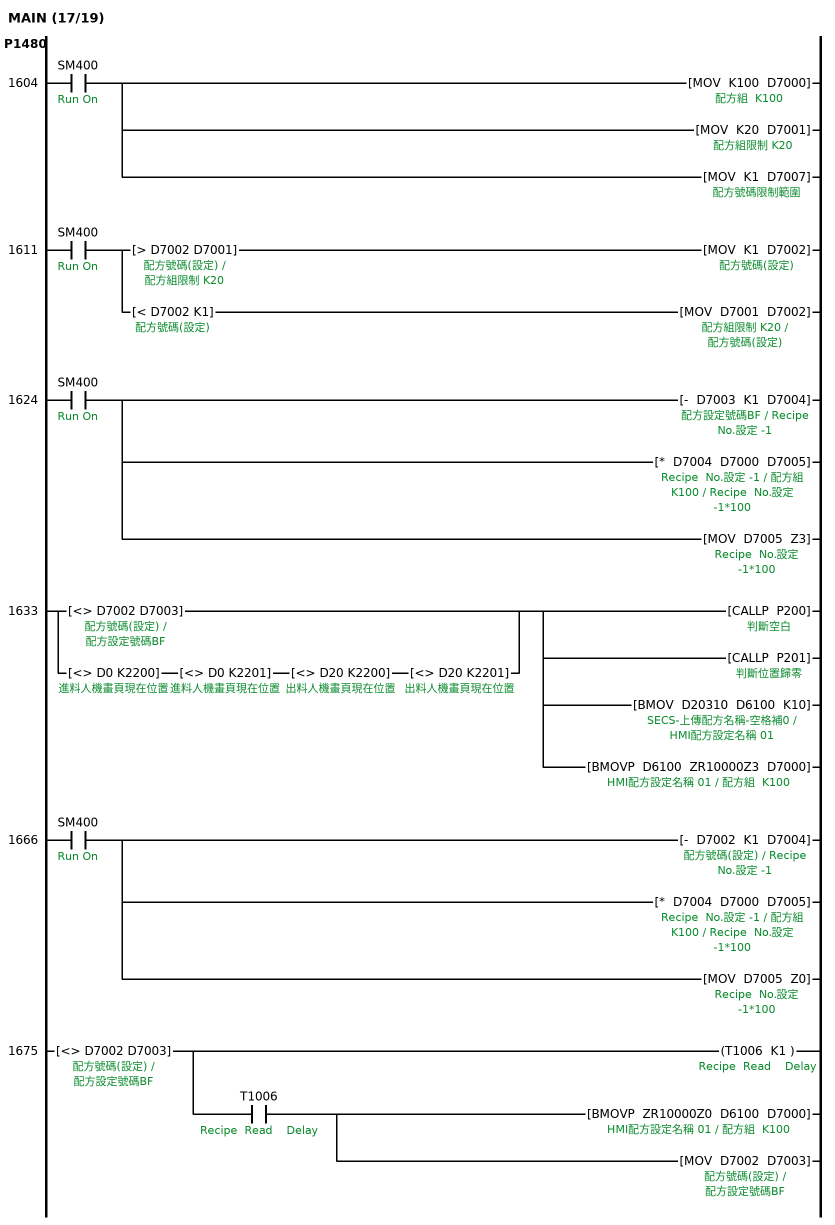
[picture p144: ladder of MAIN, rungs at steps 1604 to 1675]
1604  LD      SM400  ; Run On
      MOV     K100 D7000  ; 配方組  K100
      MOV     K20 D7001  ; 配方組限制 K20
      MOV     K1 D7007  ; 配方號碼限制範圍
1611  LD      SM400  ; Run On
      MPS
      AND>    D7002 D7001  ; 配方號碼(設定) / 配方組限制 K20
      MOV     K1 D7002
      MPP
      AND<    D7002 K1  ; 配方號碼(設定)
      MOV     D7001 D7002
1624  LD      SM400  ; Run On
      -       D7003 K1 D7004  ; 配方設定號碼BF / Recipe  No.設定 -1
      *       D7004 D7000 D7005  ; Recipe  No.設定 -1*100
      MOV     D7005 Z3
1633  LD<>    D7002 D7003  ; 配方號碼(設定) / 配方設定號碼BF
      LD<>    D0 K2200  ; 進料人機畫頁現在位置
      AND<>   D0 K2201  ; 進料人機畫頁現在位置
      AND<>   D20 K2200  ; 出料人機畫頁現在位置
      AND<>   D20 K2201  ; 出料人機畫頁現在位置
      ORB
      CALLP   P200  ; 判斷空白
      CALLP   P201  ; 判斷位置歸零
      BMOV    D20310 D6100 K10  ; SECS-上傳配方名稱-空格補0 / HMI配方設定名稱 01
      BMOVP   D6100 ZR10000Z3 D7000
1666  LD      SM400  ; Run On
      -       D7002 K1 D7004
      *       D7004 D7000 D7005
      MOV     D7005 Z0
1675  LD<>    D7002 D7003  ; 配方號碼(設定) / 配方設定號碼BF
      OUT     T1006 K1  ; Recipe  Read    Delay
      AND     T1006  ; Recipe  Read    Delay
      BMOVP   ZR10000Z0 D6100 D7000
      MOV     D7002 D7003
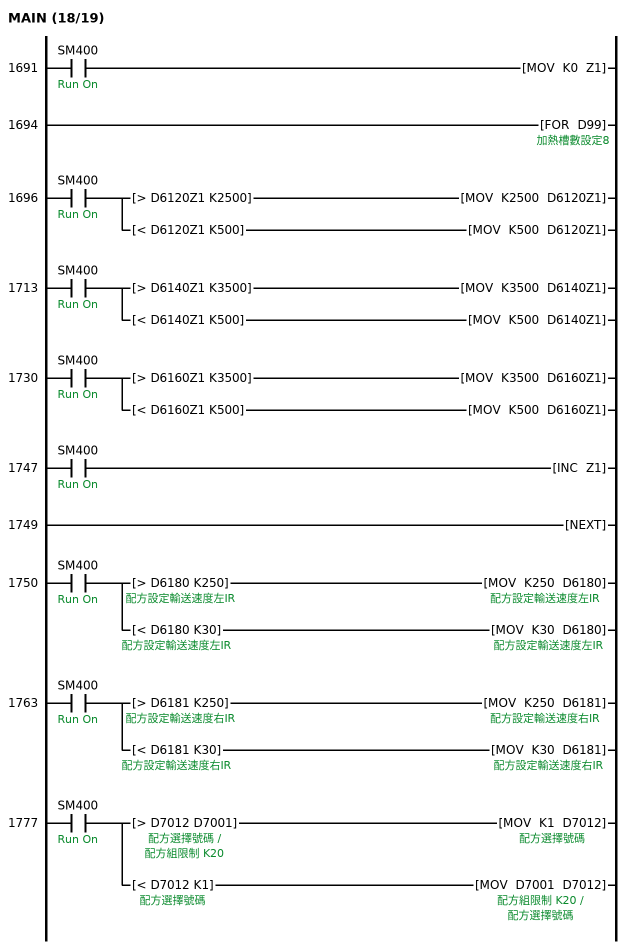
1691  LD      SM400  ; Run On
      MOV     K0 Z1
1694  FOR     D99
1696  LD      SM400  ; Run On
      MPS
      AND>    D6120Z1 K2500
      MOV     K2500 D6120Z1
      MPP
      AND<    D6120Z1 K500
      MOV     K500 D6120Z1
1713  LD      SM400  ; Run On
      MPS
      AND>    D6140Z1 K3500
      MOV     K3500 D6140Z1
      MPP
      AND<    D6140Z1 K500
      MOV     K500 D6140Z1
1730  LD      SM400  ; Run On
      MPS
      AND>    D6160Z1 K3500
      MOV     K3500 D6160Z1
      MPP
      AND<    D6160Z1 K500
      MOV     K500 D6160Z1
1747  LD      SM400  ; Run On
      INC     Z1
1749  NEXT
1750  LD      SM400  ; Run On
      MPS
      AND>    D6180 K250  ; 配方設定輸送速度左IR
      MOV     K250 D6180
      MPP
      AND<    D6180 K30  ; 配方設定輸送速度左IR
      MOV     K30 D6180
1763  LD      SM400  ; Run On
      MPS
      AND>    D6181 K250  ; 配方設定輸送速度右IR
      MOV     K250 D6181
      MPP
      AND<    D6181 K30  ; 配方設定輸送速度右IR
      MOV     K30 D6181
1777  LD      SM400  ; Run On
      MPS
      AND>    D7012 D7001  ; 配方選擇號碼 / 配方組限制 K20
      MOV     K1 D7012
      MPP
      AND<    D7012 K1  ; 配方選擇號碼
      MOV     D7001 D7012
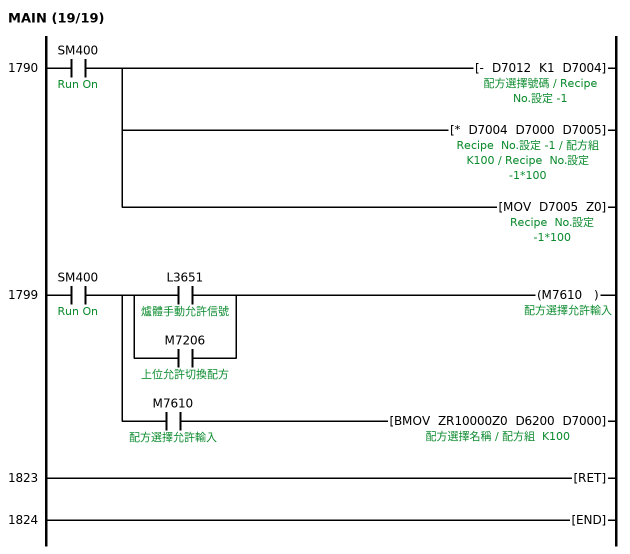
1790  LD      SM400  ; Run On
      -       D7012 K1 D7004
      *       D7004 D7000 D7005
      MOV     D7005 Z0
1799  LD      SM400  ; Run On
      MPS
      LD      L3651  ; 爐體手動允許信號
      OR      M7206  ; 上位允許切換配方
      ANB
      OUT     M7610  ; 配方選擇允許輸入
      MPP
      AND     M7610  ; 配方選擇允許輸入
      BMOV    ZR10000Z0 D6200 D7000  ; 配方選擇名稱
        [note] /* 配方選擇切換 */
1823  RET
1824  END
END_PROGRAM

PROGRAM HEAT
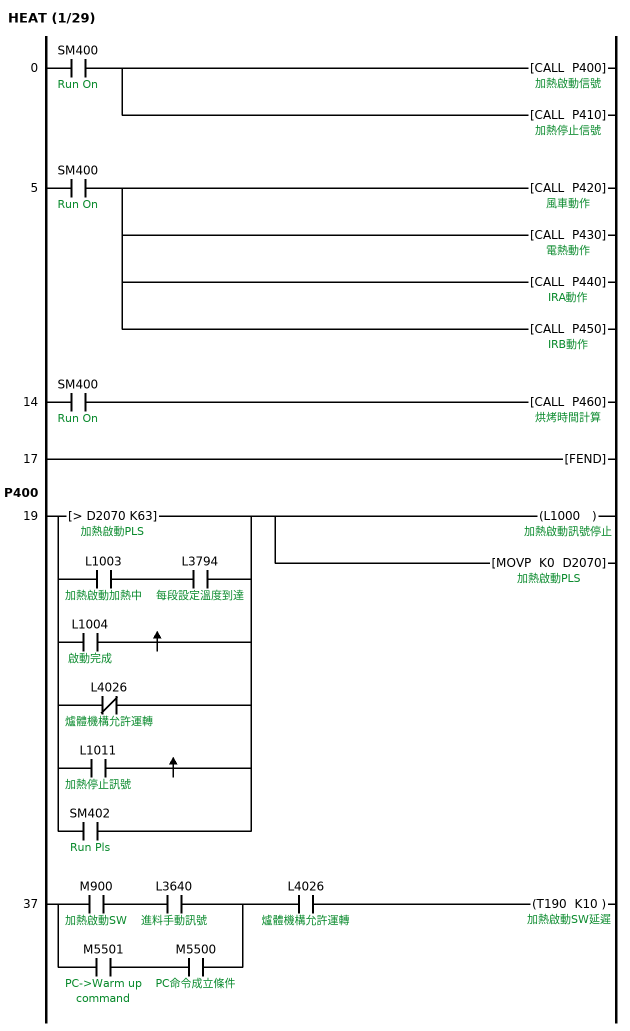
0     LD      SM400  ; Run On
      CALL    P400  ; 加熱啟動信號
      CALL    P410  ; 加熱停止信號
5     LD      SM400  ; Run On
      CALL    P420  ; 風車動作
      CALL    P430  ; 電熱動作
      CALL    P440  ; IRA動作
      CALL    P450  ; IRB動作
14    LD      SM400  ; Run On
      CALL    P460  ; 烘烤時間計算
17    FEND
      P400
19    LD>     D2070 K63  ; 加熱啟動PLS
      LD      L1003  ; 加熱啟動加熱中
      AND     L3794  ; 每段設定溫度到達
      ORB
      LD      L1004  ; 啟動完成
      MEP
      ORB
      ORI     L4026  ; 爐體機構允許運轉
      LD      L1011  ; 加熱停止訊號
      MEP
      ORB
      OR      SM402  ; Run Pls
      OUT     L1000  ; 加熱啟動訊號停止
      MOVP    K0 D2070
37    LD      M900  ; 加熱啟動SW
      AND     L3640  ; 進料手動訊號
      LD      M5501  ; PC->Warm up command
      AND     M5500  ; PC命令成立條件
      ORB
      AND     L4026  ; 爐體機構允許運轉
      OUT     T190 K10  ; 加熱啟動SW延遲
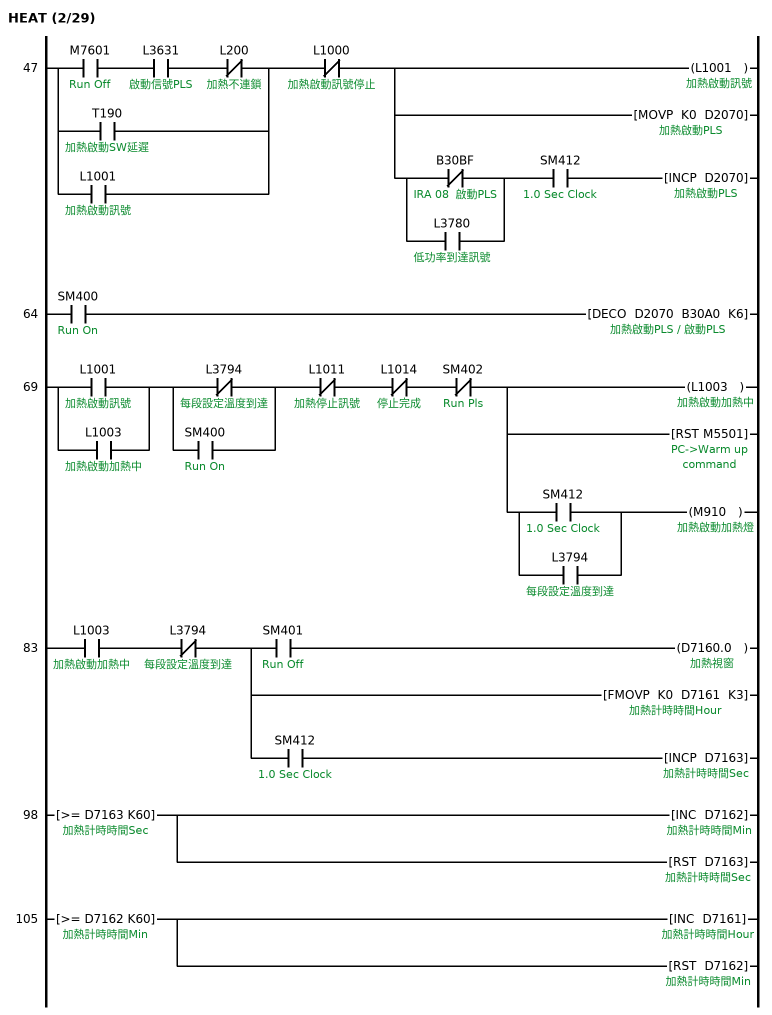
47    LD      M7601  ; Run Off
      AND     L3631  ; 啟動信號PLS
      ANI     L200  ; 加熱不連鎖
      OR      T190  ; 加熱啟動SW延遲
      OR      L1001  ; 加熱啟動訊號
      ANI     L1000  ; 加熱啟動訊號停止
      OUT     L1001  ; 加熱啟動訊號
      MOVP    K0 D2070
      LDI     B30BF  ; IRA 08  啟動PLS
      OR      L3780  ; 低功率到達訊號
      ANB
      AND     SM412  ; 1.0 Sec Clock
      INCP    D2070
64    LD      SM400  ; Run On
      DECO    D2070 B30A0 K6  ; 啟動PLS
69    LD      L1001  ; 加熱啟動訊號
      OR      L1003  ; 加熱啟動加熱中
      LDI     L3794  ; 每段設定溫度到達
      OR      SM400  ; Run On
      ANB
      ANI     L1011  ; 加熱停止訊號
      ANI     L1014  ; 停止完成
      ANI     SM402  ; Run Pls
      OUT     L1003  ; 加熱啟動加熱中
      RST     M5501  ; PC->Warm up command
      LD      SM412  ; 1.0 Sec Clock
      OR      L3794  ; 每段設定溫度到達
      ANB
      OUT     M910  ; 加熱啟動加熱燈
83    LD      L1003  ; 加熱啟動加熱中
      ANI     L3794  ; 每段設定溫度到達
      MPS
      AND     SM401  ; Run Off
      OUT     D7160.0  ; 加熱視窗
      MPP
      FMOVP   K0 D7161 K3  ; 加熱計時時間Hour
      AND     SM412  ; 1.0 Sec Clock
      INCP    D7163  ; 加熱計時時間Sec
98    LD>=    D7163 K60  ; 加熱計時時間Sec
      INC     D7162  ; 加熱計時時間Min
      RST     D7163  ; 加熱計時時間Sec
105   LD>=    D7162 K60  ; 加熱計時時間Min
      INC     D7161
      RST     D7162  ; 加熱計時時間Min
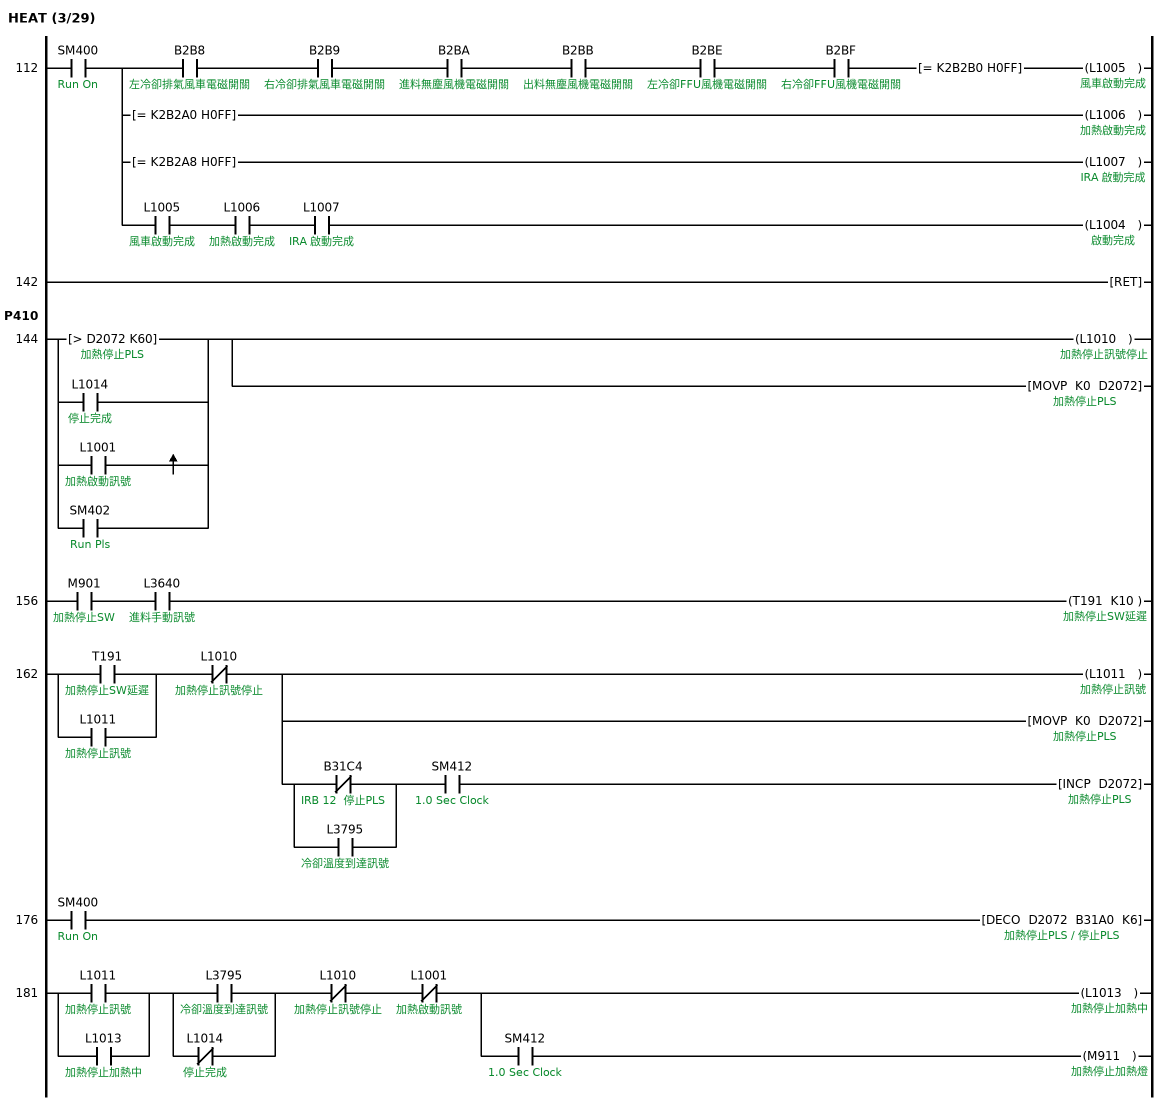
112   LD      SM400  ; Run On
      MPS
      AND     B2B8  ; 左冷卻排氣風車電磁開關
      AND     B2B9  ; 右冷卻排氣風車電磁開關
      AND     B2BA  ; 進料無塵風機電磁開關
      AND     B2BB  ; 出料無塵風機電磁開關
      AND     B2BE  ; 左冷卻FFU風機電磁開關
      AND     B2BF  ; 右冷卻FFU風機電磁開關
      AND=    K2B2B0 H0FF  ; 第01槽風車電磁開關
      OUT     L1005  ; 風車啟動完成
      MRD
      AND=    K2B2A0 H0FF  ; 第01槽熱風H01電磁開關
      OUT     L1006  ; 加熱啟動完成
      MRD
      AND=    K2B2A8 H0FF  ; 第01槽IR01A電磁開關
      OUT     L1007  ; IRA 啟動完成
      MPP
      AND     L1005  ; 風車啟動完成
      AND     L1006  ; 加熱啟動完成
      AND     L1007  ; IRA 啟動完成
      OUT     L1004  ; 啟動完成
142   RET
      P410
144   LD>     D2072 K60  ; 加熱停止PLS
      OR      L1014  ; 停止完成
      LD      L1001  ; 加熱啟動訊號
      MEP
      ORB
      OR      SM402  ; Run Pls
      OUT     L1010  ; 加熱停止訊號停止
      MOVP    K0 D2072
156   LD      M901  ; 加熱停止SW
      AND     L3640  ; 進料手動訊號
      OUT     T191 K10  ; 加熱停止SW延遲
162   LD      T191  ; 加熱停止SW延遲
      OR      L1011  ; 加熱停止訊號
      ANI     L1010  ; 加熱停止訊號停止
      OUT     L1011  ; 加熱停止訊號
      MOVP    K0 D2072
      LDI     B31C4  ; IRB 12  停止PLS
      OR      L3795  ; 冷卻溫度到達訊號
      ANB
      AND     SM412  ; 1.0 Sec Clock
      INCP    D2072
176   LD      SM400  ; Run On
      DECO    D2072 B31A0 K6  ; 停止PLS
181   LD      L1011  ; 加熱停止訊號
      OR      L1013  ; 加熱停止加熱中
      LD      L3795  ; 冷卻溫度到達訊號
      ORI     L1014  ; 停止完成
      ANB
      ANI     L1010  ; 加熱停止訊號停止
      ANI     L1001  ; 加熱啟動訊號
      OUT     L1013  ; 加熱停止加熱中
      AND     SM412  ; 1.0 Sec Clock
      OUT     M911  ; 加熱停止加熱燈
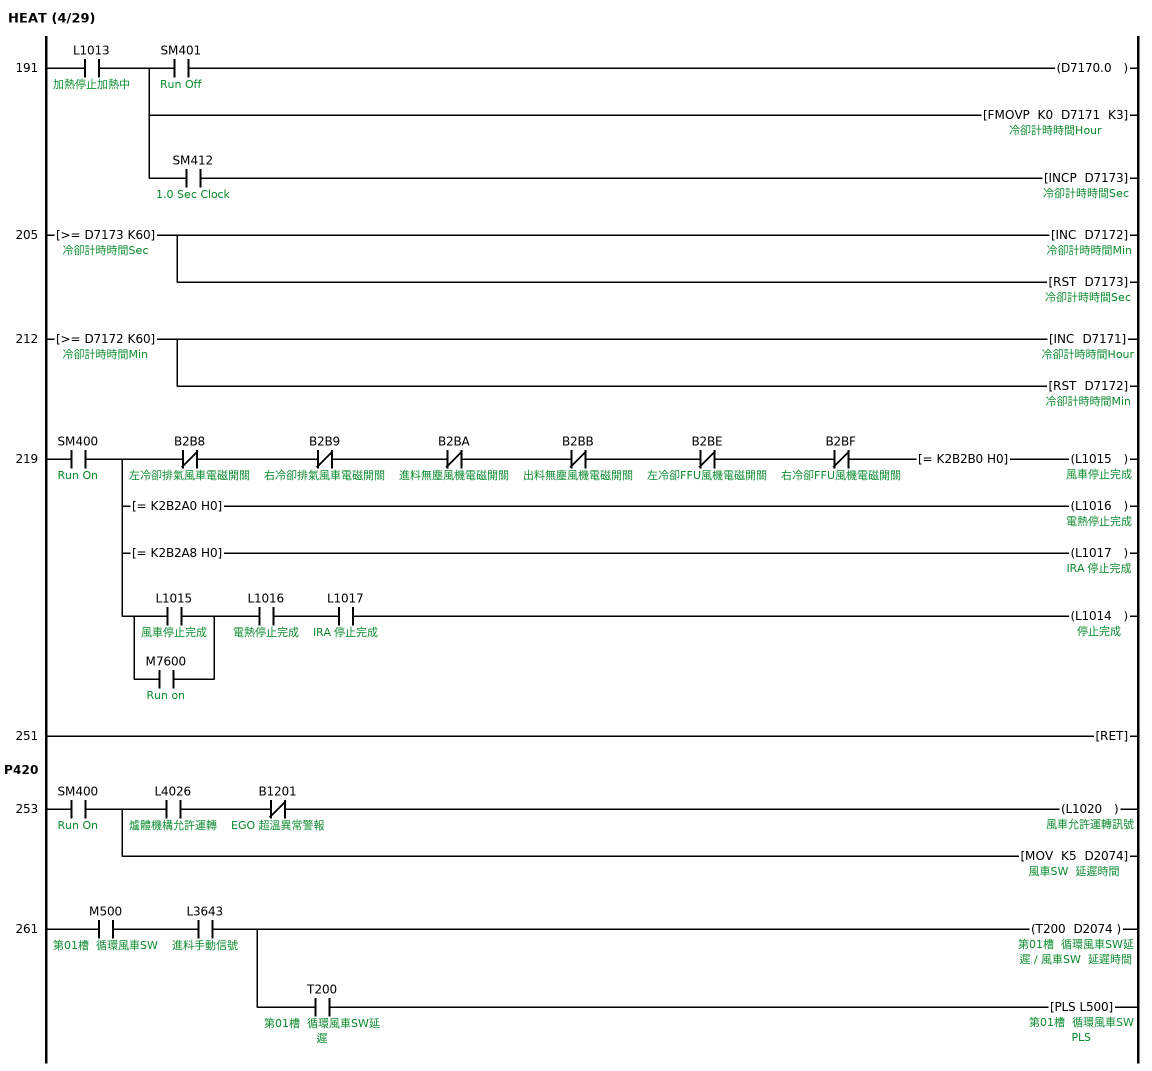
191   LD      L1013  ; 加熱停止加熱中
      MPS
      AND     SM401  ; Run Off
      OUT     D7170.0
      MPP
      FMOVP   K0 D7171 K3  ; 冷卻計時時間Hour
      AND     SM412  ; 1.0 Sec Clock
      INCP    D7173  ; 冷卻計時時間Sec
205   LD>=    D7173 K60  ; 冷卻計時時間Sec
      INC     D7172  ; 冷卻計時時間Min
      RST     D7173  ; 冷卻計時時間Sec
212   LD>=    D7172 K60  ; 冷卻計時時間Min
      INC     D7171
      RST     D7172  ; 冷卻計時時間Min
219   LD      SM400  ; Run On
      MPS
      ANI     B2B8  ; 左冷卻排氣風車電磁開關
      ANI     B2B9  ; 右冷卻排氣風車電磁開關
      ANI     B2BA  ; 進料無塵風機電磁開關
      ANI     B2BB  ; 出料無塵風機電磁開關
      ANI     B2BE  ; 左冷卻FFU風機電磁開關
      ANI     B2BF  ; 右冷卻FFU風機電磁開關
      AND=    K2B2B0 H0  ; 第01槽風車電磁開關
      OUT     L1015  ; 風車停止完成
      MRD
      AND=    K2B2A0 H0  ; 第01槽熱風H01電磁開關
      OUT     L1016  ; 電熱停止完成
      MRD
      AND=    K2B2A8 H0  ; 第01槽IR01A電磁開關
      OUT     L1017  ; IRA 停止完成
      MPP
      LD      L1015  ; 風車停止完成
      OR      M7600  ; Run on
      ANB
      AND     L1016  ; 電熱停止完成
      AND     L1017  ; IRA 停止完成
      OUT     L1014  ; 停止完成
251   RET
      P420
253   LD      SM400  ; Run On
      MPS
      AND     L4026  ; 爐體機構允許運轉
      ANI     B1201  ; EGO 超溫異常警報
      OUT     L1020  ; 風車允許運轉訊號
      MPP
      MOV     K5 D2074  ; 風車SW  延遲時間
261   LD      M500  ; 第01槽  循環風車SW
      AND     L3643  ; 進料手動信號
      OUT     T200 D2074  ; 第01槽  循環風車SW延遲 / 風車SW  延遲時間
      AND     T200  ; 第01槽  循環風車SW延遲
      PLS     L500  ; 第01槽  循環風車SW  PLS
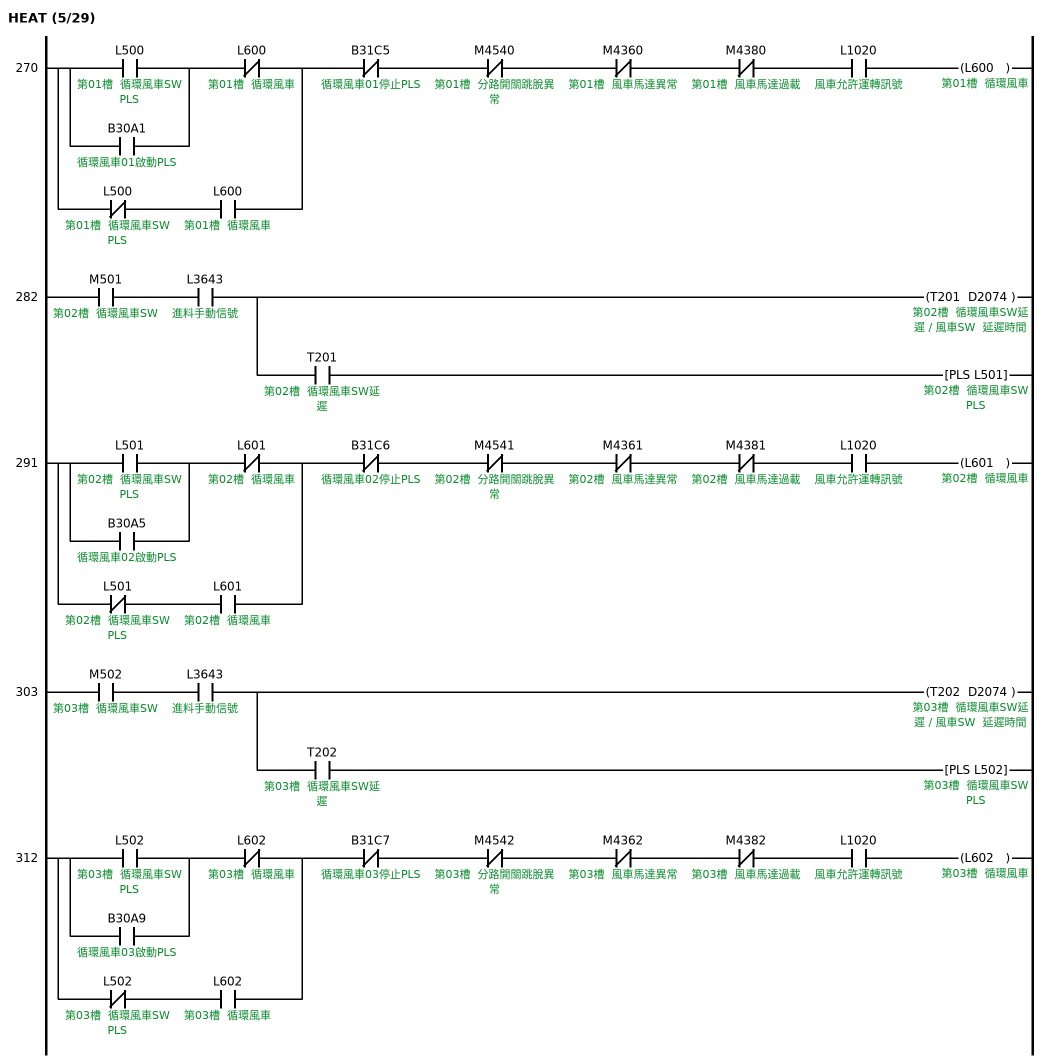
270   LD      L500  ; 第01槽  循環風車SW  PLS
      OR      B30A1  ; 循環風車01啟動PLS
      ANI     L600  ; 第01槽  循環風車
      LDI     L500  ; 第01槽  循環風車SW  PLS
      AND     L600  ; 第01槽  循環風車
      ORB
      ANI     B31C5  ; 循環風車01停止PLS
      ANI     M4540  ; 第01槽  分路開關跳脫異常
      ANI     M4360  ; 第01槽  風車馬達異常
      ANI     M4380  ; 第01槽  風車馬達過載
      AND     L1020  ; 風車允許運轉訊號
      OUT     L600  ; 第01槽  循環風車
282   LD      M501  ; 第02槽  循環風車SW
      AND     L3643  ; 進料手動信號
      OUT     T201 D2074  ; 第02槽  循環風車SW延遲 / 風車SW  延遲時間
      AND     T201  ; 第02槽  循環風車SW延遲
      PLS     L501  ; 第02槽  循環風車SW  PLS
291   LD      L501  ; 第02槽  循環風車SW  PLS
      OR      B30A5  ; 循環風車02啟動PLS
      ANI     L601  ; 第02槽  循環風車
      LDI     L501  ; 第02槽  循環風車SW  PLS
      AND     L601  ; 第02槽  循環風車
      ORB
      ANI     B31C6  ; 循環風車02停止PLS
      ANI     M4541  ; 第02槽  分路開關跳脫異常
      ANI     M4361  ; 第02槽  風車馬達異常
      ANI     M4381  ; 第02槽  風車馬達過載
      AND     L1020  ; 風車允許運轉訊號
      OUT     L601  ; 第02槽  循環風車
303   LD      M502  ; 第03槽  循環風車SW
      AND     L3643  ; 進料手動信號
      OUT     T202 D2074  ; 第03槽  循環風車SW延遲 / 風車SW  延遲時間
      AND     T202  ; 第03槽  循環風車SW延遲
      PLS     L502  ; 第03槽  循環風車SW  PLS
312   LD      L502  ; 第03槽  循環風車SW  PLS
      OR      B30A9  ; 循環風車03啟動PLS
      ANI     L602  ; 第03槽  循環風車
      LDI     L502  ; 第03槽  循環風車SW  PLS
      AND     L602  ; 第03槽  循環風車
      ORB
      ANI     B31C7  ; 循環風車03停止PLS
      ANI     M4542  ; 第03槽  分路開關跳脫異常
      ANI     M4362  ; 第03槽  風車馬達異常
      ANI     M4382  ; 第03槽  風車馬達過載
      AND     L1020  ; 風車允許運轉訊號
      OUT     L602  ; 第03槽  循環風車
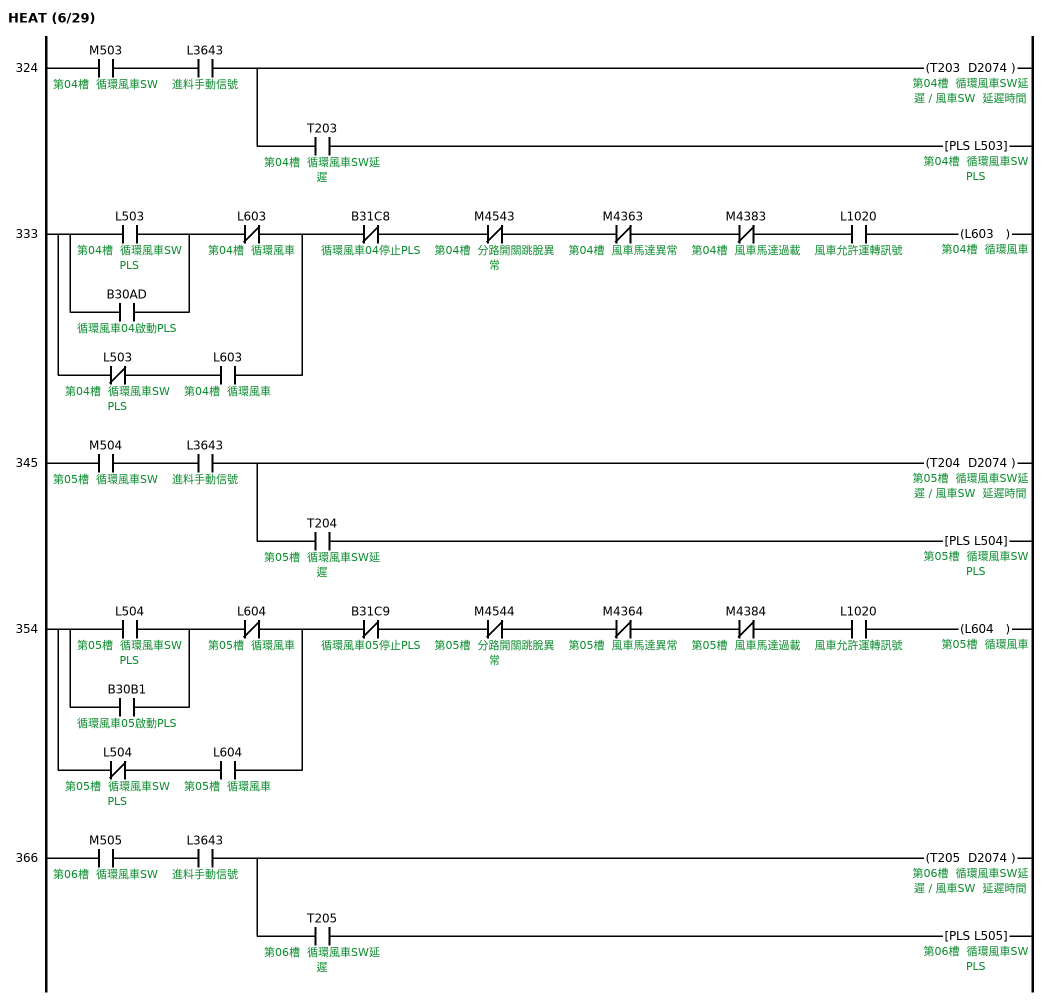
324   LD      M503  ; 第04槽  循環風車SW
      AND     L3643  ; 進料手動信號
      OUT     T203 D2074  ; 第04槽  循環風車SW延遲 / 風車SW  延遲時間
      AND     T203  ; 第04槽  循環風車SW延遲
      PLS     L503  ; 第04槽  循環風車SW  PLS
333   LD      L503  ; 第04槽  循環風車SW  PLS
      OR      B30AD  ; 循環風車04啟動PLS
      ANI     L603  ; 第04槽  循環風車
      LDI     L503  ; 第04槽  循環風車SW  PLS
      AND     L603  ; 第04槽  循環風車
      ORB
      ANI     B31C8  ; 循環風車04停止PLS
      ANI     M4543  ; 第04槽  分路開關跳脫異常
      ANI     M4363  ; 第04槽  風車馬達異常
      ANI     M4383  ; 第04槽  風車馬達過載
      AND     L1020  ; 風車允許運轉訊號
      OUT     L603  ; 第04槽  循環風車
345   LD      M504  ; 第05槽  循環風車SW
      AND     L3643  ; 進料手動信號
      OUT     T204 D2074  ; 第05槽  循環風車SW延遲 / 風車SW  延遲時間
      AND     T204  ; 第05槽  循環風車SW延遲
      PLS     L504  ; 第05槽  循環風車SW  PLS
354   LD      L504  ; 第05槽  循環風車SW  PLS
      OR      B30B1  ; 循環風車05啟動PLS
      ANI     L604  ; 第05槽  循環風車
      LDI     L504  ; 第05槽  循環風車SW  PLS
      AND     L604  ; 第05槽  循環風車
      ORB
      ANI     B31C9  ; 循環風車05停止PLS
      ANI     M4544  ; 第05槽  分路開關跳脫異常
      ANI     M4364  ; 第05槽  風車馬達異常
      ANI     M4384  ; 第05槽  風車馬達過載
      AND     L1020  ; 風車允許運轉訊號
      OUT     L604  ; 第05槽  循環風車
366   LD      M505  ; 第06槽  循環風車SW
      AND     L3643  ; 進料手動信號
      OUT     T205 D2074  ; 第06槽  循環風車SW延遲 / 風車SW  延遲時間
      AND     T205  ; 第06槽  循環風車SW延遲
      PLS     L505  ; 第06槽  循環風車SW  PLS
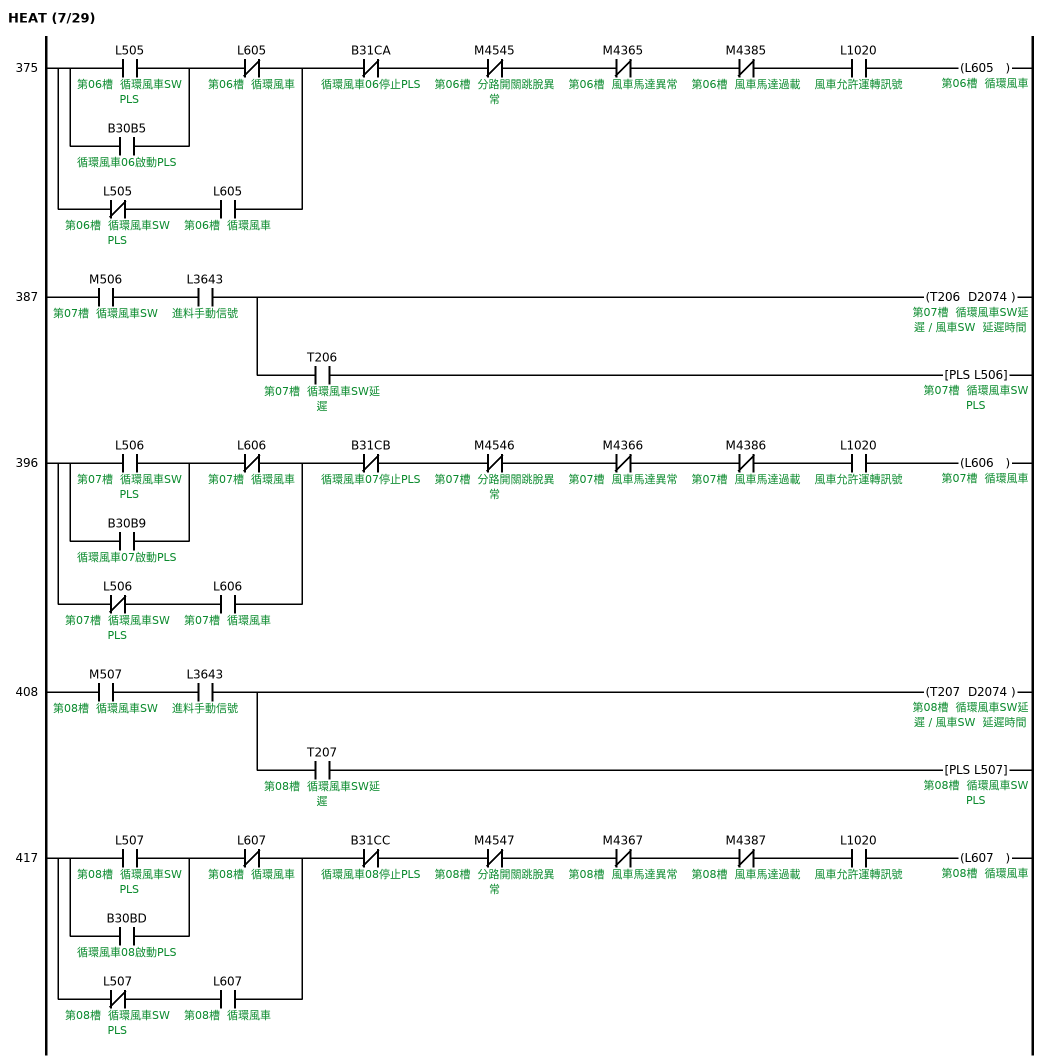
375   LD      L505  ; 第06槽  循環風車SW  PLS
      OR      B30B5  ; 循環風車06啟動PLS
      ANI     L605  ; 第06槽  循環風車
      LDI     L505  ; 第06槽  循環風車SW  PLS
      AND     L605  ; 第06槽  循環風車
      ORB
      ANI     B31CA  ; 循環風車06停止PLS
      ANI     M4545  ; 第06槽  分路開關跳脫異常
      ANI     M4365  ; 第06槽  風車馬達異常
      ANI     M4385  ; 第06槽  風車馬達過載
      AND     L1020  ; 風車允許運轉訊號
      OUT     L605  ; 第06槽  循環風車
387   LD      M506  ; 第07槽  循環風車SW
      AND     L3643  ; 進料手動信號
      OUT     T206 D2074  ; 第07槽  循環風車SW延遲 / 風車SW  延遲時間
      AND     T206  ; 第07槽  循環風車SW延遲
      PLS     L506  ; 第07槽  循環風車SW  PLS
396   LD      L506  ; 第07槽  循環風車SW  PLS
      OR      B30B9  ; 循環風車07啟動PLS
      ANI     L606  ; 第07槽  循環風車
      LDI     L506  ; 第07槽  循環風車SW  PLS
      AND     L606  ; 第07槽  循環風車
      ORB
      ANI     B31CB  ; 循環風車07停止PLS
      ANI     M4546  ; 第07槽  分路開關跳脫異常
      ANI     M4366  ; 第07槽  風車馬達異常
      ANI     M4386  ; 第07槽  風車馬達過載
      AND     L1020  ; 風車允許運轉訊號
      OUT     L606  ; 第07槽  循環風車
408   LD      M507  ; 第08槽  循環風車SW
      AND     L3643  ; 進料手動信號
      OUT     T207 D2074  ; 第08槽  循環風車SW延遲 / 風車SW  延遲時間
      AND     T207  ; 第08槽  循環風車SW延遲
      PLS     L507  ; 第08槽  循環風車SW  PLS
417   LD      L507  ; 第08槽  循環風車SW  PLS
      OR      B30BD  ; 循環風車08啟動PLS
      ANI     L607  ; 第08槽  循環風車
      LDI     L507  ; 第08槽  循環風車SW  PLS
      AND     L607  ; 第08槽  循環風車
      ORB
      ANI     B31CC  ; 循環風車08停止PLS
      ANI     M4547  ; 第08槽  分路開關跳脫異常
      ANI     M4367  ; 第08槽  風車馬達異常
      ANI     M4387  ; 第08槽  風車馬達過載
      AND     L1020  ; 風車允許運轉訊號
      OUT     L607  ; 第08槽  循環風車
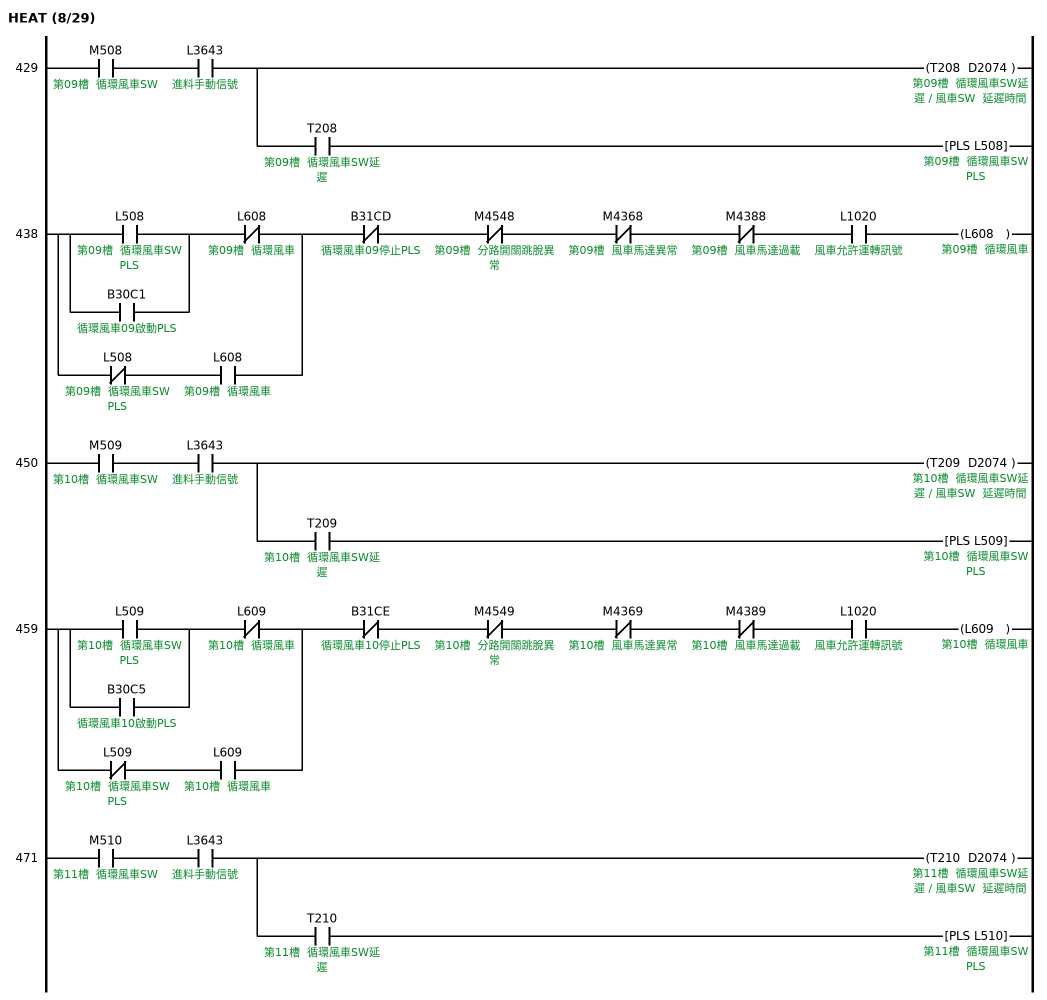
429   LD      M508  ; 第09槽  循環風車SW
      AND     L3643  ; 進料手動信號
      OUT     T208 D2074  ; 第09槽  循環風車SW延遲 / 風車SW  延遲時間
      AND     T208  ; 第09槽  循環風車SW延遲
      PLS     L508  ; 第09槽  循環風車SW  PLS
438   LD      L508  ; 第09槽  循環風車SW  PLS
      OR      B30C1  ; 循環風車09啟動PLS
      ANI     L608  ; 第09槽  循環風車
      LDI     L508  ; 第09槽  循環風車SW  PLS
      AND     L608  ; 第09槽  循環風車
      ORB
      ANI     B31CD  ; 循環風車09停止PLS
      ANI     M4548  ; 第09槽  分路開關跳脫異常
      ANI     M4368  ; 第09槽  風車馬達異常
      ANI     M4388  ; 第09槽  風車馬達過載
      AND     L1020  ; 風車允許運轉訊號
      OUT     L608  ; 第09槽  循環風車
450   LD      M509  ; 第10槽  循環風車SW
      AND     L3643  ; 進料手動信號
      OUT     T209 D2074  ; 第10槽  循環風車SW延遲 / 風車SW  延遲時間
      AND     T209  ; 第10槽  循環風車SW延遲
      PLS     L509  ; 第10槽  循環風車SW  PLS
459   LD      L509  ; 第10槽  循環風車SW  PLS
      OR      B30C5  ; 循環風車10啟動PLS
      ANI     L609  ; 第10槽  循環風車
      LDI     L509  ; 第10槽  循環風車SW  PLS
      AND     L609  ; 第10槽  循環風車
      ORB
      ANI     B31CE  ; 循環風車10停止PLS
      ANI     M4549  ; 第10槽  分路開關跳脫異常
      ANI     M4369  ; 第10槽  風車馬達異常
      ANI     M4389  ; 第10槽  風車馬達過載
      AND     L1020  ; 風車允許運轉訊號
      OUT     L609  ; 第10槽  循環風車
471   LD      M510  ; 第11槽  循環風車SW
      AND     L3643  ; 進料手動信號
      OUT     T210 D2074  ; 第11槽  循環風車SW延遲 / 風車SW  延遲時間
      AND     T210  ; 第11槽  循環風車SW延遲
      PLS     L510  ; 第11槽  循環風車SW  PLS
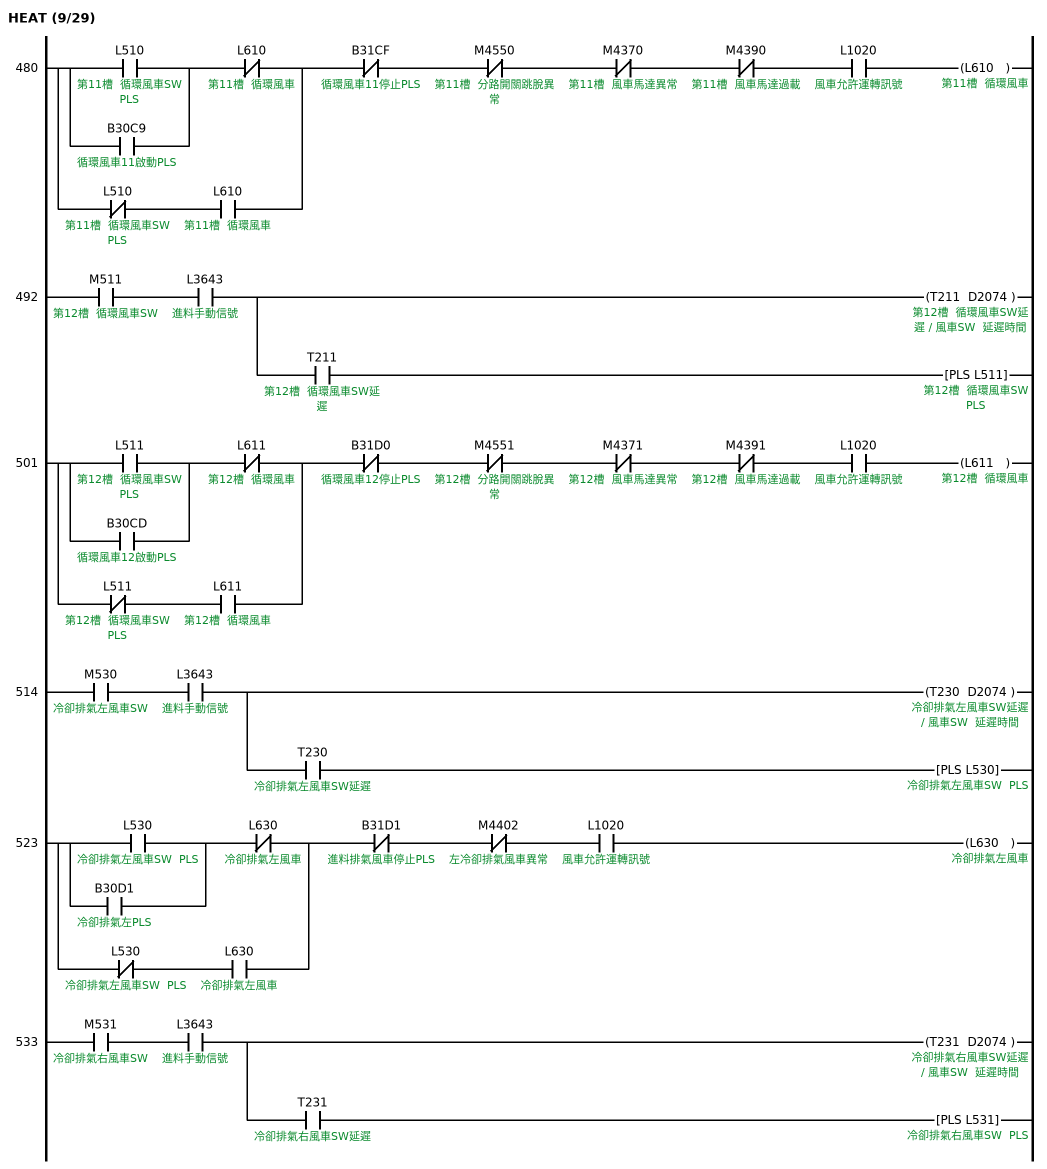
480   LD      L510  ; 第11槽  循環風車SW  PLS
      OR      B30C9  ; 循環風車11啟動PLS
      ANI     L610  ; 第11槽  循環風車
      LDI     L510  ; 第11槽  循環風車SW  PLS
      AND     L610  ; 第11槽  循環風車
      ORB
      ANI     B31CF  ; 循環風車11停止PLS
      ANI     M4550  ; 第11槽  分路開關跳脫異常
      ANI     M4370  ; 第11槽  風車馬達異常
      ANI     M4390  ; 第11槽  風車馬達過載
      AND     L1020  ; 風車允許運轉訊號
      OUT     L610  ; 第11槽  循環風車
492   LD      M511  ; 第12槽  循環風車SW
      AND     L3643  ; 進料手動信號
      OUT     T211 D2074  ; 第12槽  循環風車SW延遲 / 風車SW  延遲時間
      AND     T211  ; 第12槽  循環風車SW延遲
      PLS     L511  ; 第12槽  循環風車SW  PLS
501   LD      L511  ; 第12槽  循環風車SW  PLS
      OR      B30CD  ; 循環風車12啟動PLS
      ANI     L611  ; 第12槽  循環風車
      LDI     L511  ; 第12槽  循環風車SW  PLS
      AND     L611  ; 第12槽  循環風車
      ORB
      ANI     B31D0  ; 循環風車12停止PLS
      ANI     M4551  ; 第12槽  分路開關跳脫異常
      ANI     M4371  ; 第12槽  風車馬達異常
      ANI     M4391  ; 第12槽  風車馬達過載
      AND     L1020  ; 風車允許運轉訊號
      OUT     L611  ; 第12槽  循環風車
514   LD      M530  ; 冷卻排氣左風車SW
      AND     L3643  ; 進料手動信號
      OUT     T230 D2074  ; 冷卻排氣左風車SW延遲 / 風車SW  延遲時間
      AND     T230  ; 冷卻排氣左風車SW延遲
      PLS     L530  ; 冷卻排氣左風車SW  PLS
523   LD      L530  ; 冷卻排氣左風車SW  PLS
      OR      B30D1  ; 冷卻排氣左PLS
      ANI     L630  ; 冷卻排氣左風車
      LDI     L530  ; 冷卻排氣左風車SW  PLS
      AND     L630  ; 冷卻排氣左風車
      ORB
      ANI     B31D1  ; 進料排氣風車停止PLS
      ANI     M4402  ; 左冷卻排氣風車異常
      AND     L1020  ; 風車允許運轉訊號
      OUT     L630  ; 冷卻排氣左風車
533   LD      M531  ; 冷卻排氣右風車SW
      AND     L3643  ; 進料手動信號
      OUT     T231 D2074  ; 冷卻排氣右風車SW延遲 / 風車SW  延遲時間
      AND     T231  ; 冷卻排氣右風車SW延遲
      PLS     L531  ; 冷卻排氣右風車SW  PLS
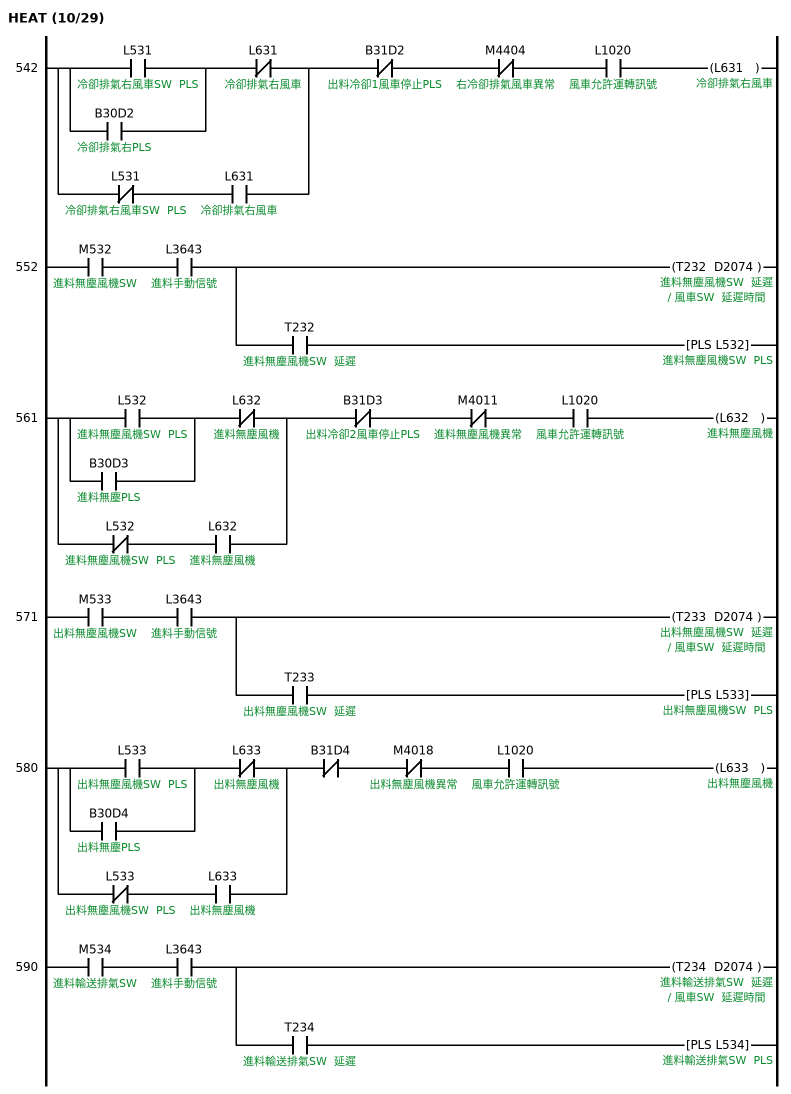
542   LD      L531  ; 冷卻排氣右風車SW  PLS
      OR      B30D2  ; 冷卻排氣右PLS
      ANI     L631  ; 冷卻排氣右風車
      LDI     L531  ; 冷卻排氣右風車SW  PLS
      AND     L631  ; 冷卻排氣右風車
      ORB
      ANI     B31D2  ; 出料冷卻1風車停止PLS
      ANI     M4404  ; 右冷卻排氣風車異常
      AND     L1020  ; 風車允許運轉訊號
      OUT     L631  ; 冷卻排氣右風車
552   LD      M532  ; 進料無塵風機SW
      AND     L3643  ; 進料手動信號
      OUT     T232 D2074  ; 進料無塵風機SW  延遲 / 風車SW  延遲時間
      AND     T232  ; 進料無塵風機SW  延遲
      PLS     L532  ; 進料無塵風機SW  PLS
561   LD      L532  ; 進料無塵風機SW  PLS
      OR      B30D3  ; 進料無塵PLS
      ANI     L632  ; 進料無塵風機
      LDI     L532  ; 進料無塵風機SW  PLS
      AND     L632  ; 進料無塵風機
      ORB
      ANI     B31D3  ; 出料冷卻2風車停止PLS
      ANI     M4011  ; 進料無塵風機異常
      AND     L1020  ; 風車允許運轉訊號
      OUT     L632  ; 進料無塵風機
571   LD      M533  ; 出料無塵風機SW
      AND     L3643  ; 進料手動信號
      OUT     T233 D2074  ; 出料無塵風機SW  延遲 / 風車SW  延遲時間
      AND     T233  ; 出料無塵風機SW  延遲
      PLS     L533  ; 出料無塵風機SW  PLS
580   LD      L533  ; 出料無塵風機SW  PLS
      OR      B30D4  ; 出料無塵PLS
      ANI     L633  ; 出料無塵風機
      LDI     L533  ; 出料無塵風機SW  PLS
      AND     L633  ; 出料無塵風機
      ORB
      ANI     B31D4
      ANI     M4018  ; 出料無塵風機異常
      AND     L1020  ; 風車允許運轉訊號
      OUT     L633  ; 出料無塵風機
590   LD      M534  ; 進料輸送排氣SW
      AND     L3643  ; 進料手動信號
      OUT     T234 D2074  ; 進料輸送排氣SW  延遲 / 風車SW  延遲時間
      AND     T234  ; 進料輸送排氣SW  延遲
      PLS     L534  ; 進料輸送排氣SW  PLS
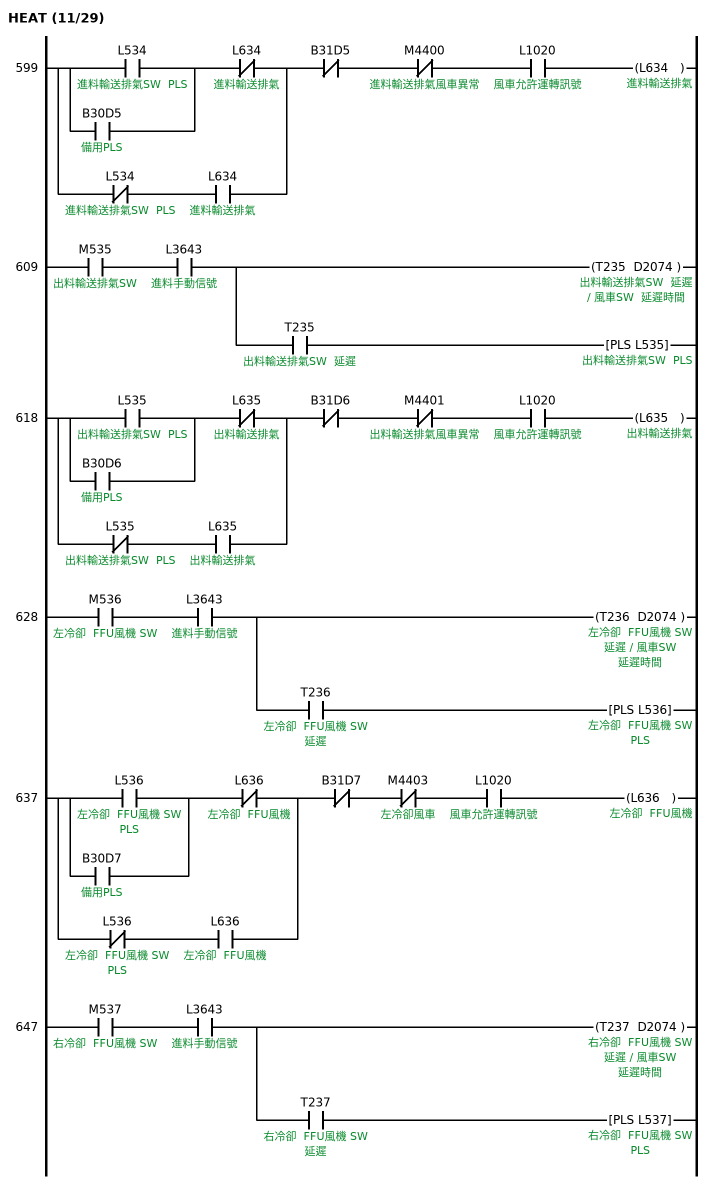
599   LD      L534  ; 進料輸送排氣SW  PLS
      OR      B30D5  ; 備用PLS
      ANI     L634  ; 進料輸送排氣
      LDI     L534  ; 進料輸送排氣SW  PLS
      AND     L634  ; 進料輸送排氣
      ORB
      ANI     B31D5
      ANI     M4400  ; 進料輸送排氣風車異常
      AND     L1020  ; 風車允許運轉訊號
      OUT     L634  ; 進料輸送排氣
609   LD      M535  ; 出料輸送排氣SW
      AND     L3643  ; 進料手動信號
      OUT     T235 D2074  ; 出料輸送排氣SW  延遲 / 風車SW  延遲時間
      AND     T235  ; 出料輸送排氣SW  延遲
      PLS     L535  ; 出料輸送排氣SW  PLS
618   LD      L535  ; 出料輸送排氣SW  PLS
      OR      B30D6  ; 備用PLS
      ANI     L635  ; 出料輸送排氣
      LDI     L535  ; 出料輸送排氣SW  PLS
      AND     L635  ; 出料輸送排氣
      ORB
      ANI     B31D6
      ANI     M4401  ; 出料輸送排氣風車異常
      AND     L1020  ; 風車允許運轉訊號
      OUT     L635  ; 出料輸送排氣
628   LD      M536  ; 左冷卻  FFU風機 SW
      AND     L3643  ; 進料手動信號
      OUT     T236 D2074  ; 左冷卻  FFU風機 SW 延遲 / 風車SW  延遲時間
      AND     T236  ; 左冷卻  FFU風機 SW 延遲
      PLS     L536  ; 左冷卻  FFU風機 SW  PLS
637   LD      L536  ; 左冷卻  FFU風機 SW  PLS
      OR      B30D7  ; 備用PLS
      ANI     L636  ; 左冷卻  FFU風機
      LDI     L536  ; 左冷卻  FFU風機 SW  PLS
      AND     L636  ; 左冷卻  FFU風機
      ORB
      ANI     B31D7
      ANI     M4403  ; 左冷卻風車
      AND     L1020  ; 風車允許運轉訊號
      OUT     L636  ; 左冷卻  FFU風機
647   LD      M537  ; 右冷卻  FFU風機 SW
      AND     L3643  ; 進料手動信號
      OUT     T237 D2074  ; 右冷卻  FFU風機 SW 延遲 / 風車SW  延遲時間
      AND     T237  ; 右冷卻  FFU風機 SW 延遲
      PLS     L537  ; 右冷卻  FFU風機 SW  PLS
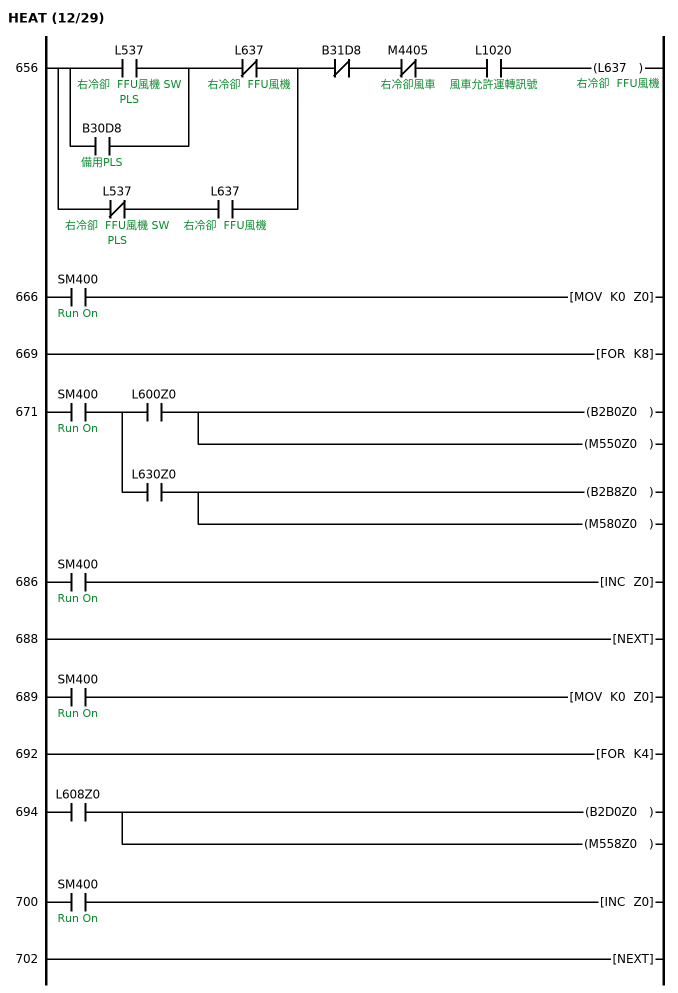
656   LD      L537  ; 右冷卻  FFU風機 SW  PLS
      OR      B30D8  ; 備用PLS
      ANI     L637  ; 右冷卻  FFU風機
      LDI     L537  ; 右冷卻  FFU風機 SW  PLS
      AND     L637  ; 右冷卻  FFU風機
      ORB
      ANI     B31D8
      ANI     M4405  ; 右冷卻風車
      AND     L1020  ; 風車允許運轉訊號
      OUT     L637  ; 右冷卻  FFU風機
666   LD      SM400  ; Run On
      MOV     K0 Z0
669   FOR     K8
671   LD      SM400  ; Run On
      MPS
      AND     L600Z0
      OUT     B2B0Z0
      OUT     M550Z0
      MPP
      AND     L630Z0
      OUT     B2B8Z0
      OUT     M580Z0
686   LD      SM400  ; Run On
      INC     Z0
688   NEXT
689   LD      SM400  ; Run On
      MOV     K0 Z0
692   FOR     K4
694   LD      L608Z0
      OUT     B2D0Z0
      OUT     M558Z0
700   LD      SM400  ; Run On
      INC     Z0
702   NEXT
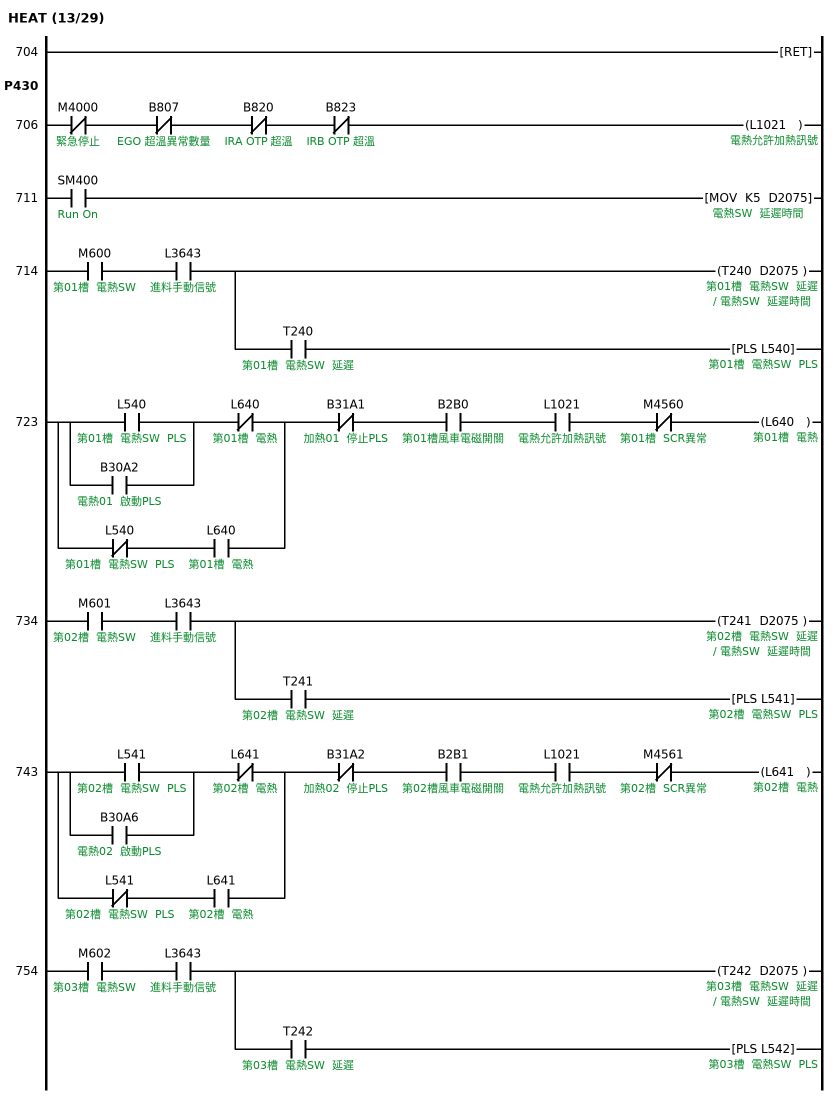
704   RET
      P430
706   LDI     M4000  ; 緊急停止
      ANI     B807  ; EGO 超溫異常數量
      ANI     B820  ; IRA OTP 超溫
      ANI     B823  ; IRB OTP 超溫
      OUT     L1021  ; 電熱允許加熱訊號
711   LD      SM400  ; Run On
      MOV     K5 D2075  ; 電熱SW  延遲時間
714   LD      M600  ; 第01槽  電熱SW
      AND     L3643  ; 進料手動信號
      OUT     T240 D2075  ; 第01槽  電熱SW  延遲 / 電熱SW  延遲時間
      AND     T240  ; 第01槽  電熱SW  延遲
      PLS     L540  ; 第01槽  電熱SW  PLS
723   LD      L540  ; 第01槽  電熱SW  PLS
      OR      B30A2  ; 電熱01  啟動PLS
      ANI     L640  ; 第01槽  電熱
      LDI     L540  ; 第01槽  電熱SW  PLS
      AND     L640  ; 第01槽  電熱
      ORB
      ANI     B31A1  ; 加熱01  停止PLS
      AND     B2B0  ; 第01槽風車電磁開關
      AND     L1021  ; 電熱允許加熱訊號
      ANI     M4560  ; 第01槽  SCR異常
      OUT     L640  ; 第01槽  電熱
734   LD      M601  ; 第02槽  電熱SW
      AND     L3643  ; 進料手動信號
      OUT     T241 D2075  ; 第02槽  電熱SW  延遲 / 電熱SW  延遲時間
      AND     T241  ; 第02槽  電熱SW  延遲
      PLS     L541  ; 第02槽  電熱SW  PLS
743   LD      L541  ; 第02槽  電熱SW  PLS
      OR      B30A6  ; 電熱02  啟動PLS
      ANI     L641  ; 第02槽  電熱
      LDI     L541  ; 第02槽  電熱SW  PLS
      AND     L641  ; 第02槽  電熱
      ORB
      ANI     B31A2  ; 加熱02  停止PLS
      AND     B2B1  ; 第02槽風車電磁開關
      AND     L1021  ; 電熱允許加熱訊號
      ANI     M4561  ; 第02槽  SCR異常
      OUT     L641  ; 第02槽  電熱
754   LD      M602  ; 第03槽  電熱SW
      AND     L3643  ; 進料手動信號
      OUT     T242 D2075  ; 第03槽  電熱SW  延遲 / 電熱SW  延遲時間
      AND     T242  ; 第03槽  電熱SW  延遲
      PLS     L542  ; 第03槽  電熱SW  PLS
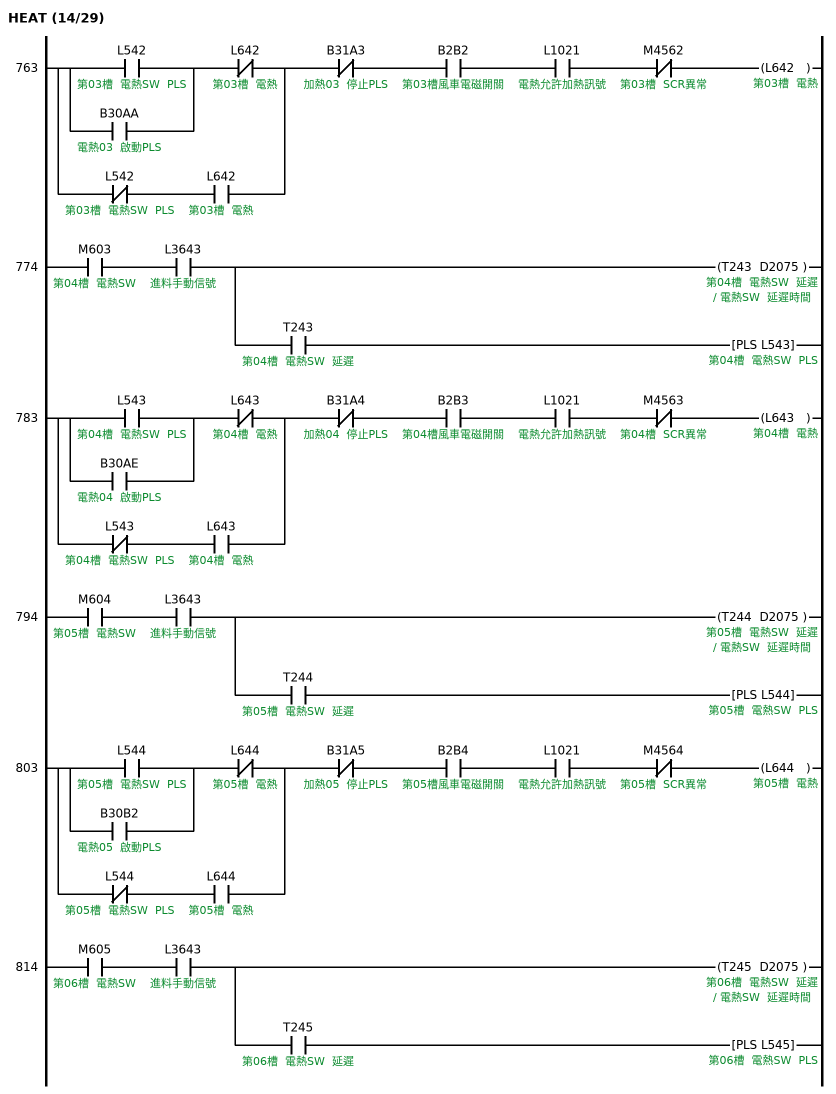
763   LD      L542  ; 第03槽  電熱SW  PLS
      OR      B30AA  ; 電熱03  啟動PLS
      ANI     L642  ; 第03槽  電熱
      LDI     L542  ; 第03槽  電熱SW  PLS
      AND     L642  ; 第03槽  電熱
      ORB
      ANI     B31A3  ; 加熱03  停止PLS
      AND     B2B2  ; 第03槽風車電磁開關
      AND     L1021  ; 電熱允許加熱訊號
      ANI     M4562  ; 第03槽  SCR異常
      OUT     L642  ; 第03槽  電熱
774   LD      M603  ; 第04槽  電熱SW
      AND     L3643  ; 進料手動信號
      OUT     T243 D2075  ; 第04槽  電熱SW  延遲 / 電熱SW  延遲時間
      AND     T243  ; 第04槽  電熱SW  延遲
      PLS     L543  ; 第04槽  電熱SW  PLS
783   LD      L543  ; 第04槽  電熱SW  PLS
      OR      B30AE  ; 電熱04  啟動PLS
      ANI     L643  ; 第04槽  電熱
      LDI     L543  ; 第04槽  電熱SW  PLS
      AND     L643  ; 第04槽  電熱
      ORB
      ANI     B31A4  ; 加熱04  停止PLS
      AND     B2B3  ; 第04槽風車電磁開關
      AND     L1021  ; 電熱允許加熱訊號
      ANI     M4563  ; 第04槽  SCR異常
      OUT     L643  ; 第04槽  電熱
794   LD      M604  ; 第05槽  電熱SW
      AND     L3643  ; 進料手動信號
      OUT     T244 D2075  ; 第05槽  電熱SW  延遲 / 電熱SW  延遲時間
      AND     T244  ; 第05槽  電熱SW  延遲
      PLS     L544  ; 第05槽  電熱SW  PLS
803   LD      L544  ; 第05槽  電熱SW  PLS
      OR      B30B2  ; 電熱05  啟動PLS
      ANI     L644  ; 第05槽  電熱
      LDI     L544  ; 第05槽  電熱SW  PLS
      AND     L644  ; 第05槽  電熱
      ORB
      ANI     B31A5  ; 加熱05  停止PLS
      AND     B2B4  ; 第05槽風車電磁開關
      AND     L1021  ; 電熱允許加熱訊號
      ANI     M4564  ; 第05槽  SCR異常
      OUT     L644  ; 第05槽  電熱
814   LD      M605  ; 第06槽  電熱SW
      AND     L3643  ; 進料手動信號
      OUT     T245 D2075  ; 第06槽  電熱SW  延遲 / 電熱SW  延遲時間
      AND     T245  ; 第06槽  電熱SW  延遲
      PLS     L545  ; 第06槽  電熱SW  PLS
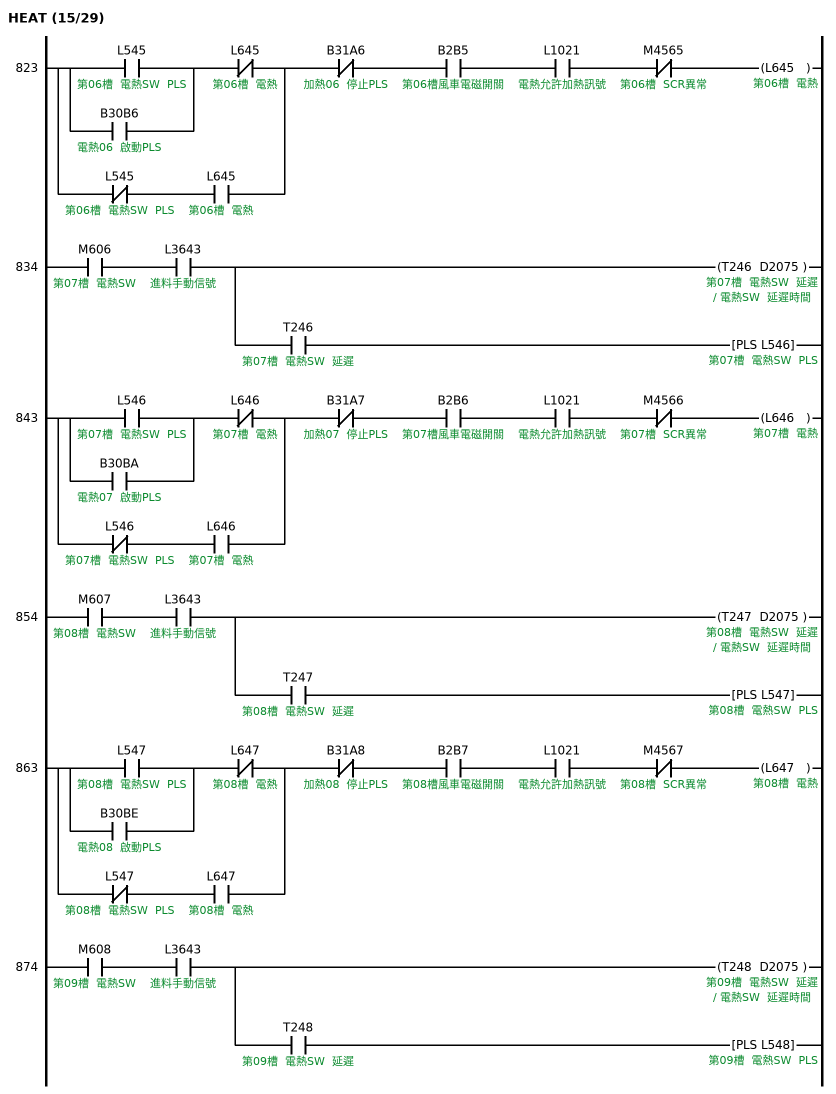
823   LD      L545  ; 第06槽  電熱SW  PLS
      OR      B30B6  ; 電熱06  啟動PLS
      ANI     L645  ; 第06槽  電熱
      LDI     L545  ; 第06槽  電熱SW  PLS
      AND     L645  ; 第06槽  電熱
      ORB
      ANI     B31A6  ; 加熱06  停止PLS
      AND     B2B5  ; 第06槽風車電磁開關
      AND     L1021  ; 電熱允許加熱訊號
      ANI     M4565  ; 第06槽  SCR異常
      OUT     L645  ; 第06槽  電熱
834   LD      M606  ; 第07槽  電熱SW
      AND     L3643  ; 進料手動信號
      OUT     T246 D2075  ; 第07槽  電熱SW  延遲 / 電熱SW  延遲時間
      AND     T246  ; 第07槽  電熱SW  延遲
      PLS     L546  ; 第07槽  電熱SW  PLS
843   LD      L546  ; 第07槽  電熱SW  PLS
      OR      B30BA  ; 電熱07  啟動PLS
      ANI     L646  ; 第07槽  電熱
      LDI     L546  ; 第07槽  電熱SW  PLS
      AND     L646  ; 第07槽  電熱
      ORB
      ANI     B31A7  ; 加熱07  停止PLS
      AND     B2B6  ; 第07槽風車電磁開關
      AND     L1021  ; 電熱允許加熱訊號
      ANI     M4566  ; 第07槽  SCR異常
      OUT     L646  ; 第07槽  電熱
854   LD      M607  ; 第08槽  電熱SW
      AND     L3643  ; 進料手動信號
      OUT     T247 D2075  ; 第08槽  電熱SW  延遲 / 電熱SW  延遲時間
      AND     T247  ; 第08槽  電熱SW  延遲
      PLS     L547  ; 第08槽  電熱SW  PLS
863   LD      L547  ; 第08槽  電熱SW  PLS
      OR      B30BE  ; 電熱08  啟動PLS
      ANI     L647  ; 第08槽  電熱
      LDI     L547  ; 第08槽  電熱SW  PLS
      AND     L647  ; 第08槽  電熱
      ORB
      ANI     B31A8  ; 加熱08  停止PLS
      AND     B2B7  ; 第08槽風車電磁開關
      AND     L1021  ; 電熱允許加熱訊號
      ANI     M4567  ; 第08槽  SCR異常
      OUT     L647  ; 第08槽  電熱
874   LD      M608  ; 第09槽  電熱SW
      AND     L3643  ; 進料手動信號
      OUT     T248 D2075  ; 第09槽  電熱SW  延遲 / 電熱SW  延遲時間
      AND     T248  ; 第09槽  電熱SW  延遲
      PLS     L548  ; 第09槽  電熱SW  PLS
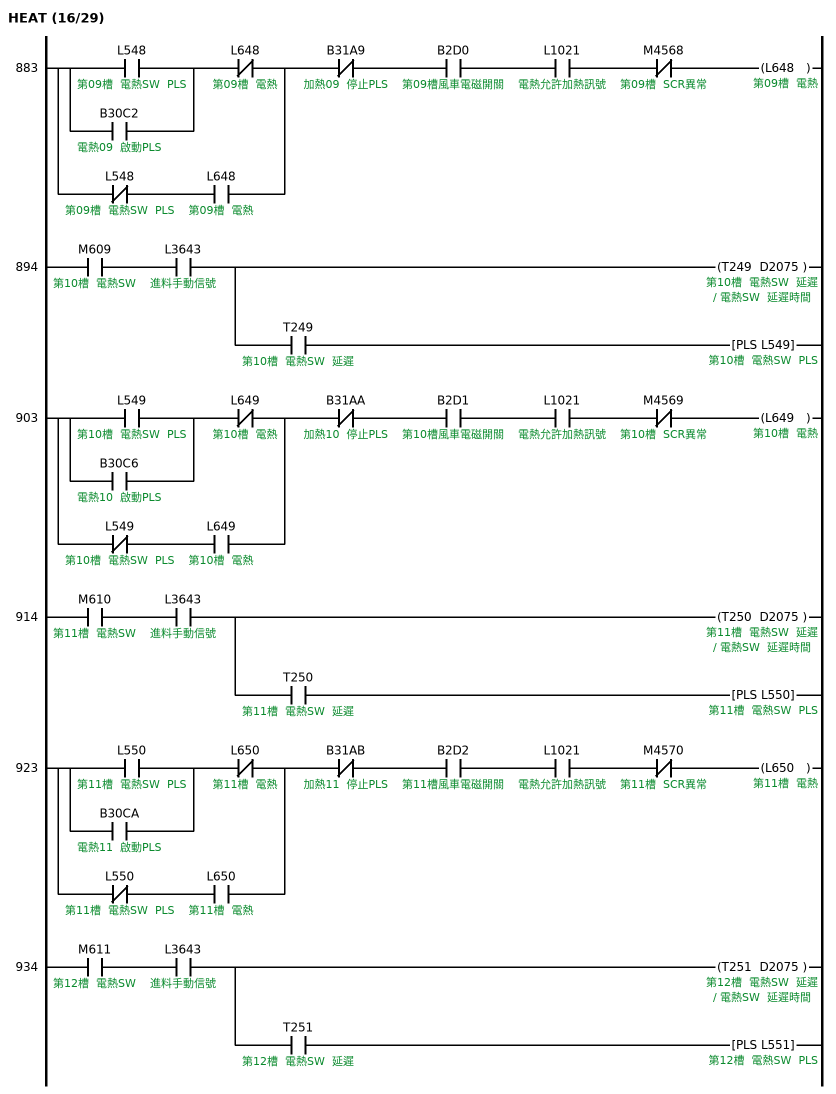
883   LD      L548  ; 第09槽  電熱SW  PLS
      OR      B30C2  ; 電熱09  啟動PLS
      ANI     L648  ; 第09槽  電熱
      LDI     L548  ; 第09槽  電熱SW  PLS
      AND     L648  ; 第09槽  電熱
      ORB
      ANI     B31A9  ; 加熱09  停止PLS
      AND     B2D0  ; 第09槽風車電磁開關
      AND     L1021  ; 電熱允許加熱訊號
      ANI     M4568  ; 第09槽  SCR異常
      OUT     L648  ; 第09槽  電熱
894   LD      M609  ; 第10槽  電熱SW
      AND     L3643  ; 進料手動信號
      OUT     T249 D2075  ; 第10槽  電熱SW  延遲 / 電熱SW  延遲時間
      AND     T249  ; 第10槽  電熱SW  延遲
      PLS     L549  ; 第10槽  電熱SW  PLS
903   LD      L549  ; 第10槽  電熱SW  PLS
      OR      B30C6  ; 電熱10  啟動PLS
      ANI     L649  ; 第10槽  電熱
      LDI     L549  ; 第10槽  電熱SW  PLS
      AND     L649  ; 第10槽  電熱
      ORB
      ANI     B31AA  ; 加熱10  停止PLS
      AND     B2D1  ; 第10槽風車電磁開關
      AND     L1021  ; 電熱允許加熱訊號
      ANI     M4569  ; 第10槽  SCR異常
      OUT     L649  ; 第10槽  電熱
914   LD      M610  ; 第11槽  電熱SW
      AND     L3643  ; 進料手動信號
      OUT     T250 D2075  ; 第11槽  電熱SW  延遲 / 電熱SW  延遲時間
      AND     T250  ; 第11槽  電熱SW  延遲
      PLS     L550  ; 第11槽  電熱SW  PLS
923   LD      L550  ; 第11槽  電熱SW  PLS
      OR      B30CA  ; 電熱11  啟動PLS
      ANI     L650  ; 第11槽  電熱
      LDI     L550  ; 第11槽  電熱SW  PLS
      AND     L650  ; 第11槽  電熱
      ORB
      ANI     B31AB  ; 加熱11  停止PLS
      AND     B2D2  ; 第11槽風車電磁開關
      AND     L1021  ; 電熱允許加熱訊號
      ANI     M4570  ; 第11槽  SCR異常
      OUT     L650  ; 第11槽  電熱
934   LD      M611  ; 第12槽  電熱SW
      AND     L3643  ; 進料手動信號
      OUT     T251 D2075  ; 第12槽  電熱SW  延遲 / 電熱SW  延遲時間
      AND     T251  ; 第12槽  電熱SW  延遲
      PLS     L551  ; 第12槽  電熱SW  PLS
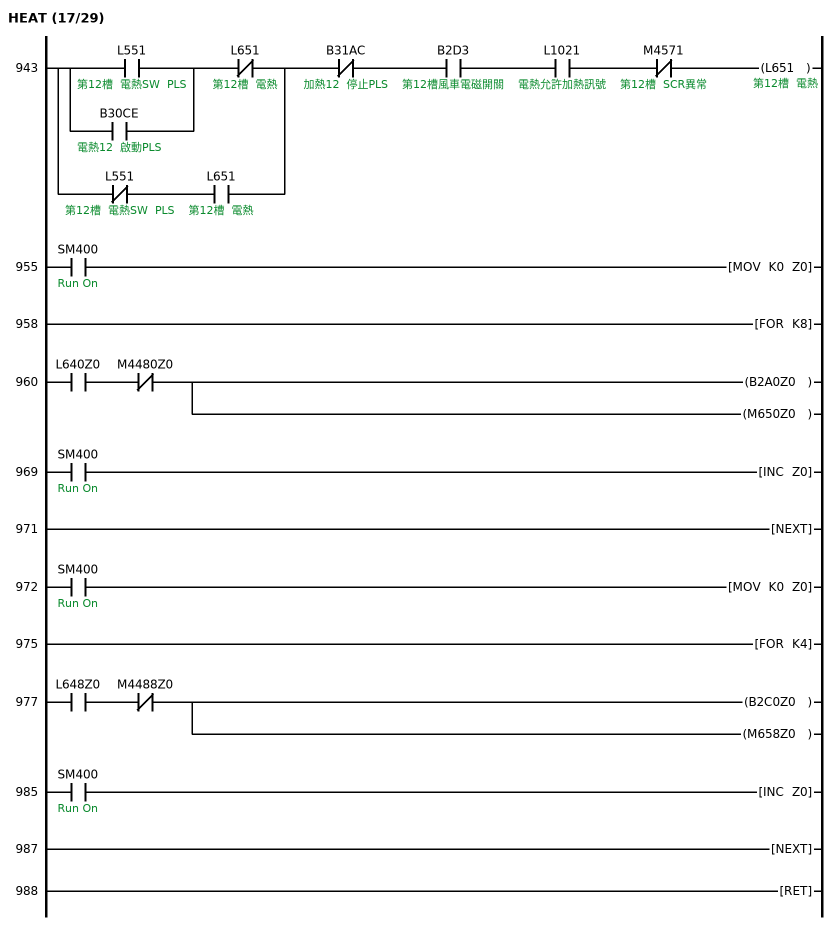
943   LD      L551  ; 第12槽  電熱SW  PLS
      OR      B30CE  ; 電熱12  啟動PLS
      ANI     L651  ; 第12槽  電熱
      LDI     L551  ; 第12槽  電熱SW  PLS
      AND     L651  ; 第12槽  電熱
      ORB
      ANI     B31AC  ; 加熱12  停止PLS
      AND     B2D3  ; 第12槽風車電磁開關
      AND     L1021  ; 電熱允許加熱訊號
      ANI     M4571  ; 第12槽  SCR異常
      OUT     L651  ; 第12槽  電熱
955   LD      SM400  ; Run On
      MOV     K0 Z0
958   FOR     K8
960   LD      L640Z0
      ANI     M4480Z0
      OUT     B2A0Z0
      OUT     M650Z0
969   LD      SM400  ; Run On
      INC     Z0
971   NEXT
972   LD      SM400  ; Run On
      MOV     K0 Z0
975   FOR     K4
977   LD      L648Z0
      ANI     M4488Z0
      OUT     B2C0Z0
      OUT     M658Z0
985   LD      SM400  ; Run On
      INC     Z0
987   NEXT
988   RET
      P440
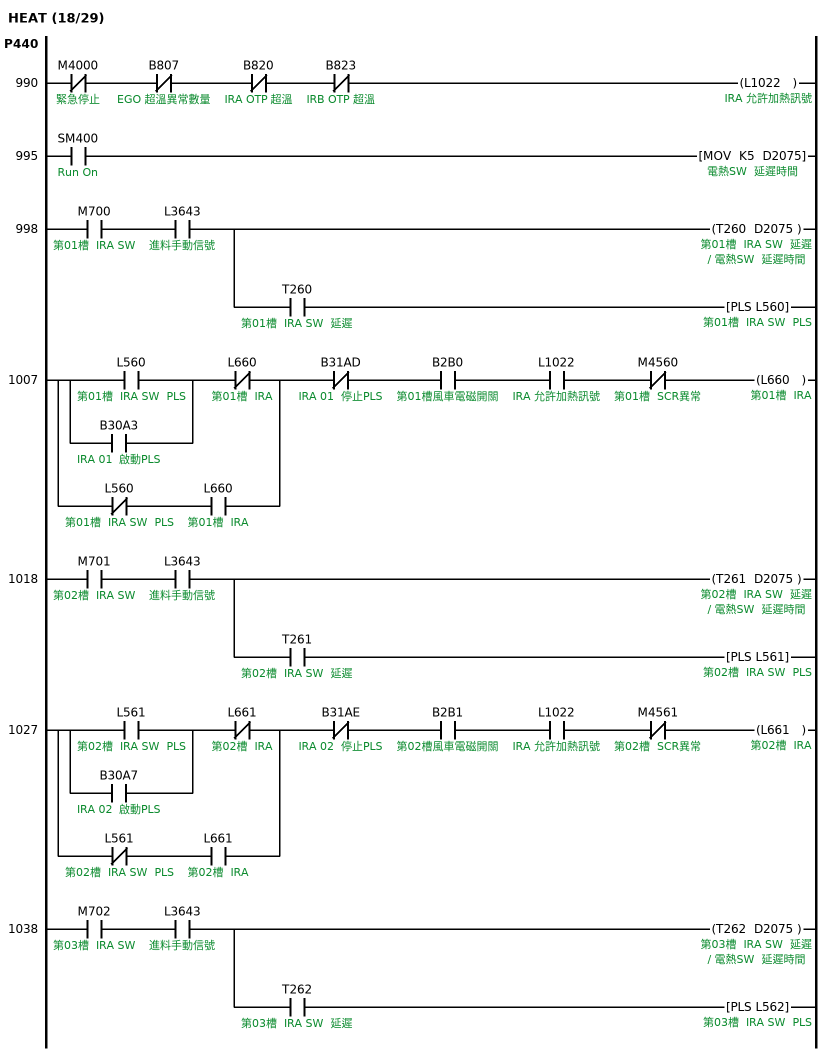
990   LDI     M4000  ; 緊急停止
      ANI     B807  ; EGO 超溫異常數量
      ANI     B820  ; IRA OTP 超溫
      ANI     B823  ; IRB OTP 超溫
      OUT     L1022  ; IRA 允許加熱訊號
995   LD      SM400  ; Run On
      MOV     K5 D2075
998   LD      M700  ; 第01槽  IRA SW
      AND     L3643  ; 進料手動信號
      OUT     T260 D2075  ; 第01槽  IRA SW  延遲 / 電熱SW  延遲時間
      AND     T260  ; 第01槽  IRA SW  延遲
      PLS     L560  ; 第01槽  IRA SW  PLS
1007  LD      L560  ; 第01槽  IRA SW  PLS
      OR      B30A3  ; IRA 01  啟動PLS
      ANI     L660  ; 第01槽  IRA
      LDI     L560  ; 第01槽  IRA SW  PLS
      AND     L660  ; 第01槽  IRA
      ORB
      ANI     B31AD  ; IRA 01  停止PLS
      AND     B2B0  ; 第01槽風車電磁開關
      AND     L1022  ; IRA 允許加熱訊號
      ANI     M4560  ; 第01槽  SCR異常
      OUT     L660  ; 第01槽  IRA
1018  LD      M701  ; 第02槽  IRA SW
      AND     L3643  ; 進料手動信號
      OUT     T261 D2075  ; 第02槽  IRA SW  延遲 / 電熱SW  延遲時間
      AND     T261  ; 第02槽  IRA SW  延遲
      PLS     L561  ; 第02槽  IRA SW  PLS
1027  LD      L561  ; 第02槽  IRA SW  PLS
      OR      B30A7  ; IRA 02  啟動PLS
      ANI     L661  ; 第02槽  IRA
      LDI     L561  ; 第02槽  IRA SW  PLS
      AND     L661  ; 第02槽  IRA
      ORB
      ANI     B31AE  ; IRA 02  停止PLS
      AND     B2B1  ; 第02槽風車電磁開關
      AND     L1022  ; IRA 允許加熱訊號
      ANI     M4561  ; 第02槽  SCR異常
      OUT     L661  ; 第02槽  IRA
1038  LD      M702  ; 第03槽  IRA SW
      AND     L3643  ; 進料手動信號
      OUT     T262 D2075  ; 第03槽  IRA SW  延遲 / 電熱SW  延遲時間
      AND     T262  ; 第03槽  IRA SW  延遲
      PLS     L562  ; 第03槽  IRA SW  PLS
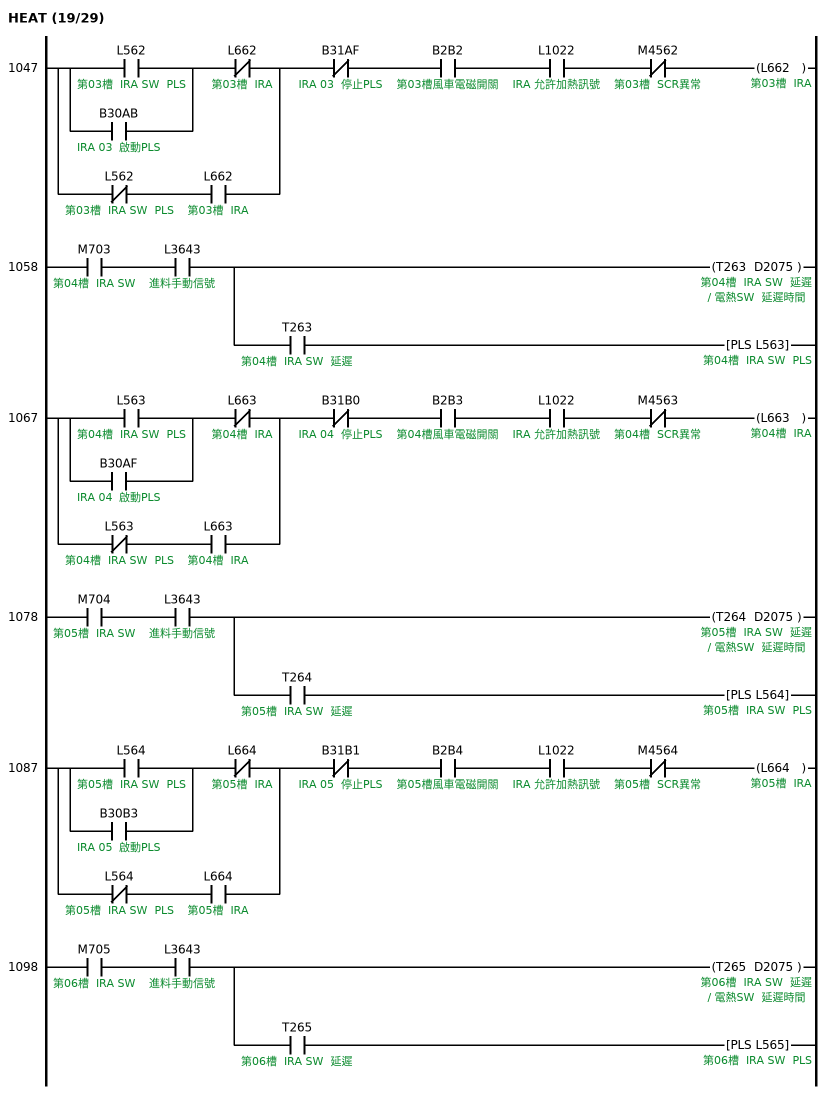
1047  LD      L562  ; 第03槽  IRA SW  PLS
      OR      B30AB  ; IRA 03  啟動PLS
      ANI     L662  ; 第03槽  IRA
      LDI     L562  ; 第03槽  IRA SW  PLS
      AND     L662  ; 第03槽  IRA
      ORB
      ANI     B31AF  ; IRA 03  停止PLS
      AND     B2B2  ; 第03槽風車電磁開關
      AND     L1022  ; IRA 允許加熱訊號
      ANI     M4562  ; 第03槽  SCR異常
      OUT     L662  ; 第03槽  IRA
1058  LD      M703  ; 第04槽  IRA SW
      AND     L3643  ; 進料手動信號
      OUT     T263 D2075  ; 第04槽  IRA SW  延遲 / 電熱SW  延遲時間
      AND     T263  ; 第04槽  IRA SW  延遲
      PLS     L563  ; 第04槽  IRA SW  PLS
1067  LD      L563  ; 第04槽  IRA SW  PLS
      OR      B30AF  ; IRA 04  啟動PLS
      ANI     L663  ; 第04槽  IRA
      LDI     L563  ; 第04槽  IRA SW  PLS
      AND     L663  ; 第04槽  IRA
      ORB
      ANI     B31B0  ; IRA 04  停止PLS
      AND     B2B3  ; 第04槽風車電磁開關
      AND     L1022  ; IRA 允許加熱訊號
      ANI     M4563  ; 第04槽  SCR異常
      OUT     L663  ; 第04槽  IRA
1078  LD      M704  ; 第05槽  IRA SW
      AND     L3643  ; 進料手動信號
      OUT     T264 D2075  ; 第05槽  IRA SW  延遲 / 電熱SW  延遲時間
      AND     T264  ; 第05槽  IRA SW  延遲
      PLS     L564  ; 第05槽  IRA SW  PLS
1087  LD      L564  ; 第05槽  IRA SW  PLS
      OR      B30B3  ; IRA 05  啟動PLS
      ANI     L664  ; 第05槽  IRA
      LDI     L564  ; 第05槽  IRA SW  PLS
      AND     L664  ; 第05槽  IRA
      ORB
      ANI     B31B1  ; IRA 05  停止PLS
      AND     B2B4  ; 第05槽風車電磁開關
      AND     L1022  ; IRA 允許加熱訊號
      ANI     M4564  ; 第05槽  SCR異常
      OUT     L664  ; 第05槽  IRA
1098  LD      M705  ; 第06槽  IRA SW
      AND     L3643  ; 進料手動信號
      OUT     T265 D2075  ; 第06槽  IRA SW  延遲 / 電熱SW  延遲時間
      AND     T265  ; 第06槽  IRA SW  延遲
      PLS     L565  ; 第06槽  IRA SW  PLS
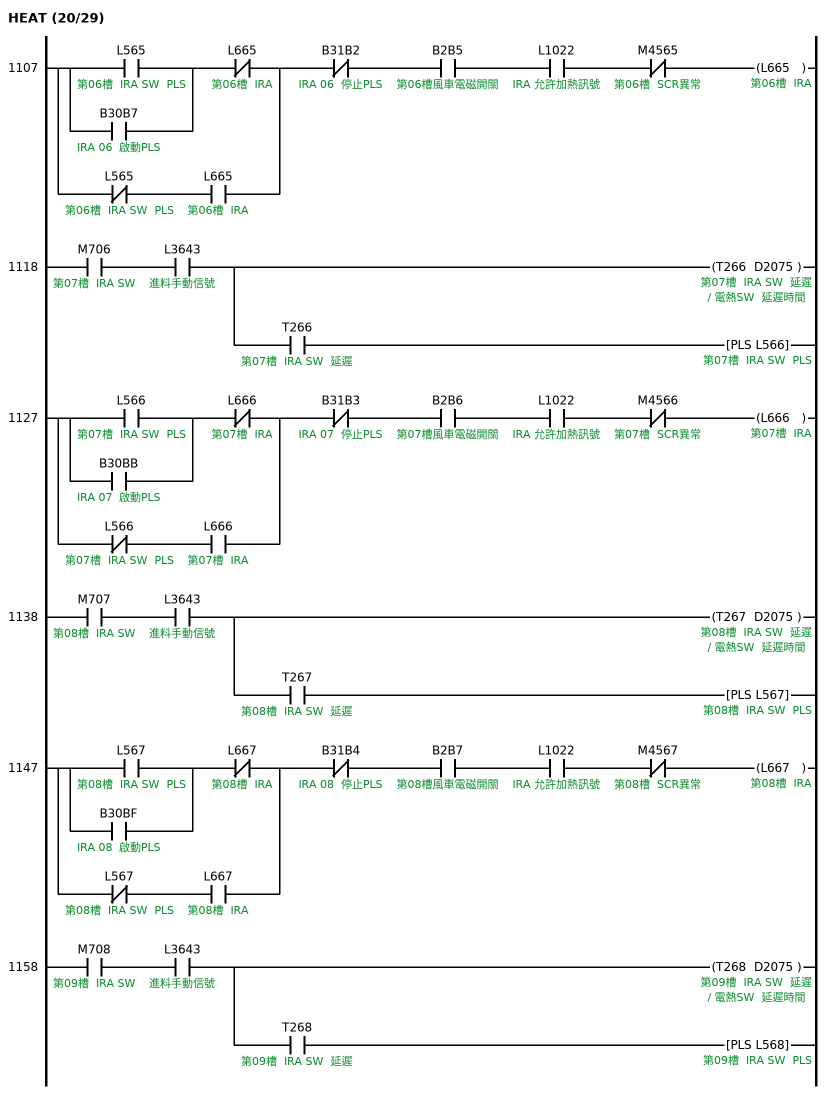
1107  LD      L565  ; 第06槽  IRA SW  PLS
      OR      B30B7  ; IRA 06  啟動PLS
      ANI     L665  ; 第06槽  IRA
      LDI     L565  ; 第06槽  IRA SW  PLS
      AND     L665  ; 第06槽  IRA
      ORB
      ANI     B31B2  ; IRA 06  停止PLS
      AND     B2B5  ; 第06槽風車電磁開關
      AND     L1022  ; IRA 允許加熱訊號
      ANI     M4565  ; 第06槽  SCR異常
      OUT     L665  ; 第06槽  IRA
1118  LD      M706  ; 第07槽  IRA SW
      AND     L3643  ; 進料手動信號
      OUT     T266 D2075  ; 第07槽  IRA SW  延遲 / 電熱SW  延遲時間
      AND     T266  ; 第07槽  IRA SW  延遲
      PLS     L566  ; 第07槽  IRA SW  PLS
1127  LD      L566  ; 第07槽  IRA SW  PLS
      OR      B30BB  ; IRA 07  啟動PLS
      ANI     L666  ; 第07槽  IRA
      LDI     L566  ; 第07槽  IRA SW  PLS
      AND     L666  ; 第07槽  IRA
      ORB
      ANI     B31B3  ; IRA 07  停止PLS
      AND     B2B6  ; 第07槽風車電磁開關
      AND     L1022  ; IRA 允許加熱訊號
      ANI     M4566  ; 第07槽  SCR異常
      OUT     L666  ; 第07槽  IRA
1138  LD      M707  ; 第08槽  IRA SW
      AND     L3643  ; 進料手動信號
      OUT     T267 D2075  ; 第08槽  IRA SW  延遲 / 電熱SW  延遲時間
      AND     T267  ; 第08槽  IRA SW  延遲
      PLS     L567  ; 第08槽  IRA SW  PLS
1147  LD      L567  ; 第08槽  IRA SW  PLS
      OR      B30BF  ; IRA 08  啟動PLS
      ANI     L667  ; 第08槽  IRA
      LDI     L567  ; 第08槽  IRA SW  PLS
      AND     L667  ; 第08槽  IRA
      ORB
      ANI     B31B4  ; IRA 08  停止PLS
      AND     B2B7  ; 第08槽風車電磁開關
      AND     L1022  ; IRA 允許加熱訊號
      ANI     M4567  ; 第08槽  SCR異常
      OUT     L667  ; 第08槽  IRA
1158  LD      M708  ; 第09槽  IRA SW
      AND     L3643  ; 進料手動信號
      OUT     T268 D2075  ; 第09槽  IRA SW  延遲 / 電熱SW  延遲時間
      AND     T268  ; 第09槽  IRA SW  延遲
      PLS     L568  ; 第09槽  IRA SW  PLS
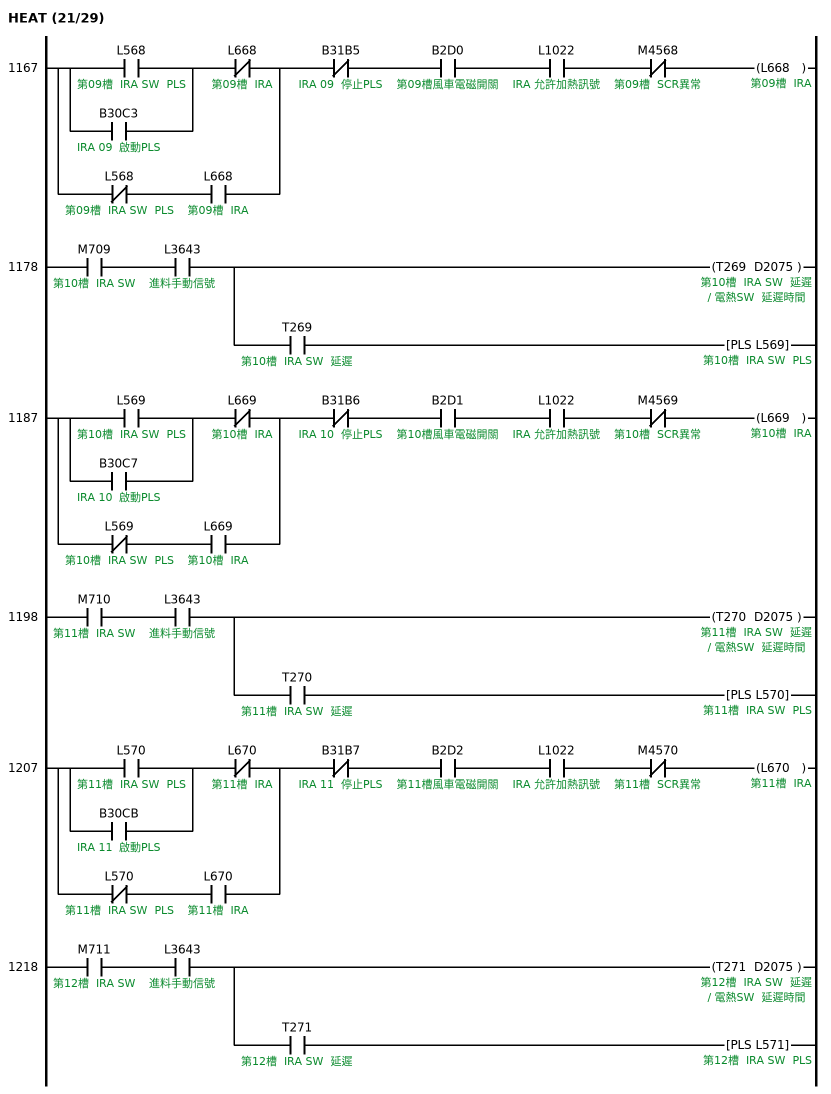
1167  LD      L568  ; 第09槽  IRA SW  PLS
      OR      B30C3  ; IRA 09  啟動PLS
      ANI     L668  ; 第09槽  IRA
      LDI     L568  ; 第09槽  IRA SW  PLS
      AND     L668  ; 第09槽  IRA
      ORB
      ANI     B31B5  ; IRA 09  停止PLS
      AND     B2D0  ; 第09槽風車電磁開關
      AND     L1022  ; IRA 允許加熱訊號
      ANI     M4568  ; 第09槽  SCR異常
      OUT     L668  ; 第09槽  IRA
1178  LD      M709  ; 第10槽  IRA SW
      AND     L3643  ; 進料手動信號
      OUT     T269 D2075  ; 第10槽  IRA SW  延遲 / 電熱SW  延遲時間
      AND     T269  ; 第10槽  IRA SW  延遲
      PLS     L569  ; 第10槽  IRA SW  PLS
1187  LD      L569  ; 第10槽  IRA SW  PLS
      OR      B30C7  ; IRA 10  啟動PLS
      ANI     L669  ; 第10槽  IRA
      LDI     L569  ; 第10槽  IRA SW  PLS
      AND     L669  ; 第10槽  IRA
      ORB
      ANI     B31B6  ; IRA 10  停止PLS
      AND     B2D1  ; 第10槽風車電磁開關
      AND     L1022  ; IRA 允許加熱訊號
      ANI     M4569  ; 第10槽  SCR異常
      OUT     L669  ; 第10槽  IRA
1198  LD      M710  ; 第11槽  IRA SW
      AND     L3643  ; 進料手動信號
      OUT     T270 D2075  ; 第11槽  IRA SW  延遲 / 電熱SW  延遲時間
      AND     T270  ; 第11槽  IRA SW  延遲
      PLS     L570  ; 第11槽  IRA SW  PLS
1207  LD      L570  ; 第11槽  IRA SW  PLS
      OR      B30CB  ; IRA 11  啟動PLS
      ANI     L670  ; 第11槽  IRA
      LDI     L570  ; 第11槽  IRA SW  PLS
      AND     L670  ; 第11槽  IRA
      ORB
      ANI     B31B7  ; IRA 11  停止PLS
      AND     B2D2  ; 第11槽風車電磁開關
      AND     L1022  ; IRA 允許加熱訊號
      ANI     M4570  ; 第11槽  SCR異常
      OUT     L670  ; 第11槽  IRA
1218  LD      M711  ; 第12槽  IRA SW
      AND     L3643  ; 進料手動信號
      OUT     T271 D2075  ; 第12槽  IRA SW  延遲 / 電熱SW  延遲時間
      AND     T271  ; 第12槽  IRA SW  延遲
      PLS     L571  ; 第12槽  IRA SW  PLS
